NameNo.	CaEVNo.	ConnectDustVacuo	:=	61	;	//
NameNo.	CaEVNo.	LineSceneDustBlow	:=	62	;	//
NameNo.  CaEVNo.	LineSceneDustVacuo	:=	63	;	//
NameNo.	CaEVNo.	AreaArrayDustBlow	:=	64	;	//
NameNo.	CaEVNo.	MouldUpBlow	:=	65	;	//
NameNo.	CaEVNo.	MouldDownVacuo	:=	66	;	//
NameNo.	CaEVNo.	MouldDownAir	:=	67	;	//
NameNo.	CaEVNo.	NGPushInsideAir	:=	68	;	//
NameNo.	CaEVNo.	NGPushInsideVacuo	:=	69	;	//
NameNo.	CaEVNo.	BrushDustVacuo_U	:=	70	;	//
NameNo.	CaEVNo.	WindDustBlow_U	:=	71	;	//
NameNo.	CaEVNo.	WindDustVacuo_U	:=	72	;	//
NameNo.	CaEVNo.	BrushDustVacuo_D	:=	73	;	//
NameNo.	CaEVNo.	WindDustBlow_D	:=	74	;	//
NameNo.	CaEVNo.	WindDustVacuo_D	:=	75	;	//
NameNo.	CaEVNo.	RJ_Blow	:=	76	;	//
NameNo.	CaEVNo.	RJDustBlow	:=	77	;	//
						
	//////纠偏号//////					
NameNo.	AnRecNo.PoleWind:=1;(***极片放卷纠偏*)					
NameNo.	AnRecNo.PoleProcess:=2;(***极片行进纠偏*)					
						
NameNo.	CaRecNo.PoleWind:=3;(***极片放卷纠偏*)					
NameNo.	CaRecNo.PoleProcess:=4;(***极片行进纠偏*)					
						
	//////凸轮编号//////					
NameNo.	AnTableNo.	Cuter	:=	11	;(*裁切切刀凸轮编号*)	
NameNo.	AnTableNo.	CuterStop	:=	12	;(*裁切切刀停止凸轮编号*)	
NameNo.	AnTableNo.	Mould	:=13	;(*模具切刀凸轮编号*)		
NameNo.	AnTableNo.	MouldStop	:=14	;(*模具切刀停止凸轮编号*)		
NameNo.	AnTableNo.	Dirver	:=15	;(*主驱动凸轮编号*)		
NameNo.	AnTableNo.	VirBelt	:=	16	;(*虚拟皮带凸轮编号*)	
NameNo.	AnTableNo.	NgPush	:=	17	;(*NG踢料凸轮编号*)	
NameNo.	AnTableNo.	NgPushStop	:=	18	;(*NG踢料停止凸轮编号*)	
NameNo.	AnTableNo.	BufferLine	:=19	;(*极片缓存凸轮编号*)		
NameNo.	AnTableNo.	CCDPress	:=	20	;(*CCD压片凸轮编号*)	
NameNo.	AnTableNo.	BufferLine_1	:=	21	;(*极片缓存凸轮编号1*)	
NameNo.	AnTableNo.VirDirver	:=	22	;(*正极虚拟驱动凸轮编号1*)	
						
NameNo.	CaTableNo.	Cuter	:=	31	;(*裁切切刀凸轮编号*)	
NameNo.	CaTableNo.	CuterStop	:=	32	;(*裁切切刀停止凸轮编号*)	
NameNo.	CaTableNo.	Mould	:=	33	;(*模具切刀凸轮编号*)	
NameNo.	CaTableNo.	MouldStop	:=	34	;(*模具切刀停止凸轮编号*)	
NameNo.	CaTableNo.	Dirver	:=	35	;(*主驱动凸轮编号*)	
NameNo.	CaTableNo.	VirBelt	:=	36	;(*虚拟皮带凸轮编号*)	
NameNo.	CaTableNo.	NgPush	:=	37	;(*NG踢料凸轮编号*)	
NameNo.	CaTableNo.	NgPushStop	:=	38	;(*NG踢料停止凸轮编号*)	
NameNo.	CaTableNo.	BufferLine	:=	39	;(*极片缓存凸轮编号*)	
NameNo.	CaTableNo.	CCDPress	:=	40	;(*CCD压片凸轮编号*)	
NameNo.	CaTableNo.	BufferLine_1	:=	41	;(*极片缓存凸轮编号1*)					
NameNo.	CaTableNo.VirDirver	:=	42	;(*负极虚拟驱动凸轮编号1*)						
	//////皮带工位号//////					
NameNo.	AnBeltNo.	First	:=1	;	//	首片数据
NameNo.	AnBeltNo.	OverHang	:=2	;	//	尺寸检测工位
NameNo.	AnBeltNo.	NGBox1	:=4	;	//	踢废工位1（连续）
NameNo.	AnBeltNo.	NGBox2	:=6	;	//	踢废工位2（单片）
NameNo.	AnBeltNo.	BrushDustU	:=7	;	//	极片上表面毛刷除尘工位
NameNo.	AnBeltNo.	WindDustU	:=8	;	//	极片上表面风刀除尘工位
NameNo.	AnBeltNo.	BrushDustD	:=9	;	//	极片下表面毛刷除尘工位
NameNo.	AnBeltNo.	WindDustD	:=10	;	//	极片下表面风刀除尘工位(除尘倒装皮带末位)
NameNo.	AnBeltNo.	SubBelt1	:=14	;	//	分段皮带1取料工位
NameNo.	AnBeltNo.	SubBelt2	:=22	;	//	分段皮带2取料工位
NameNo.	AnBeltNo.	SubBelt3	:=30	;	//	分段皮带3取料工位
						
NameNo.	CaBeltNo.	First	:=1	;	//	首片
NameNo.	CaBeltNo.	OverHang	:=2	;	//	尺寸检测工位
NameNo.	CaBeltNo.	NGBox1	:=4	;	//	踢废工位1（连续）
NameNo.	CaBeltNo.	NGBox2	:=6	;	//	踢废工位2（单片）
NameNo.	CaBeltNo.	BrushDustU	:=7	;	//	极片上表面毛刷除尘工位
NameNo.	CaBeltNo.	WindDustU	:=8	;	//	极片上表面风刀除尘工位
NameNo.	CaBeltNo.	BrushDustD	:=9	;	//	极片下表面毛刷除尘工位
NameNo.	CaBeltNo.	WindDustD	:=10	;	//	极片下表面风刀除尘工位(除尘倒装皮带末位)
NameNo.	CaBeltNo.	SubBelt1	:=12	;	//	分段皮带1取料工位
NameNo.	CaBeltNo.	SubBelt2	:=20	;	//	分段皮带2取料工位
NameNo.	CaBeltNo.	SubBelt3	:=28	;	//	分段皮带3取料工位
						
	//////极耳工位号//////					
NameNo.	AnTabNo.MouldPhoto	:=1	;	//	倒角前拍照位置	
NameNo.	AnTabNo.CuterPhoto	:=6	;	//	裁切前拍照位置	
						
NameNo.	CaTabNo.MouldPhoto	:=1	;	//	倒角前拍照位置	
NameNo.	CaTabNo.CuterPhoto	:=6	;	//	裁切前拍照位置	
						
	//////极耳间距工位号//////					
NameNo.	AnIntervalNo.First	:=1	;	//	蓝胶位置	
NameNo.	AnIntervalNo.Mould	:=5	;	//	冲R角位置	
NameNo.	AnIntervalNo.Cuter	:=10	;	//	裁切位置	
						
NameNo.	CaIntervalNo.First	:=1	;	//	蓝胶位置	
NameNo.	CaIntervalNo.Mould	:=5	;	//	冲R角位置	
NameNo.	CaIntervalNo.Cuter	:=10	;	//	裁切位置	
						
	//////除尘电机号//////	
NameNo.	AnMotorNo.	DDR_Dust	:=	1	;	//主驱辊除尘				
NameNo.	AnMotorNo.	CuterBeltDust	:=	2	;	//裁切输送皮带除尘
NameNo.	AnMotorNo.	NGReverseBeltDust	:=	3	;	//踢废倒装皮带除尘
NameNo.	AnMotorNo.	DedustBeltDust	:=	4	;	//极片上表面除尘皮带除尘
NameNo.	AnMotorNo.	DedustReverseBeltDust	:=	5	;	//极片下表面除尘倒装皮带除尘
NameNo.	AnMotorNo.	PoleBrushDust_U	:=	6	;	//极片上表面毛刷除尘
NameNo.	AnMotorNo.	PoleBrushDust_D	:=	7	;	//极片下表面毛刷除尘
NameNo.	AnMotorNo.	FeduanbeltDust1	:= 15;//正极分段皮带1毛刷
NameNo.	AnMotorNo.	FeduanbeltDust2	:= 16;//正极分段皮带2毛刷
NameNo.	AnMotorNo.	FeduanbeltDust3	:= 17;//正极分段皮带3毛刷

NameNo.	CaMotorNo.	DDR_Dust	:=	8	;	//主驱辊除尘							
NameNo.	CaMotorNo.	CuterBeltDust	:=	9	;	//裁切输送皮带除尘
NameNo.	CaMotorNo.	NGReverseBeltDust	:=	10	;	//踢废倒装皮带除尘
NameNo.	CaMotorNo.	DedustBeltDust	:=	11	;	//极片上表面除尘皮带除尘
NameNo.	CaMotorNo.	DedustReverseBeltDust	:=	12	;	//极片下表面除尘倒装皮带除尘
NameNo.	CaMotorNo.	PoleBrushDust_U	:=	13	;	//极片上表面毛刷除尘
NameNo.	CaMotorNo.	PoleBrushDust_D	:=	14	;	//极片下表面毛刷除尘
NameNo.	CaMotorNo.	FeduanbeltDust1	:=	18	;	//负极分段皮带1毛刷
NameNo.	CaMotorNo.	FeduanbeltDust2	:=	19	;	//负极分段皮带2毛刷
NameNo.	CaMotorNo.	FeduanbeltDust3	:=	20	;	//负极分段皮带3毛刷

IF ProductPar.parPublic.fMainPos <>250 THEN
	ProductPar.parPublic.fMainPos:=250;
END_IF
IF ProductPar.AnPar.fPoleWidth=0 THEN
	ProductPar.AnPar.fPoleWidth:=186;
END_IF
IF ProductPar.CaPar.fPoleWidth=0 THEN
	ProductPar.CaPar.fPoleWidth:=188;
END_IF
IF ProductPar.AnPar.Machine.fMQDriverDiameter=0 THEN
	ProductPar.AnPar.Machine.fMQDriverDiameter:=71.62;
END_IF
IF ProductPar.CaPar.Machine.fMQDriverDiameter=0 THEN
	ProductPar.CaPar.Machine.fMQDriverDiameter:=71.62;
END_IF
IF ProductPar.AnPar.iMainVel=0 THEN
	ProductPar.AnPar.iMainVel:=10;
END_IF
IF ProductPar.CaPar.iMainVel=0 THEN
	ProductPar.CaPar.iMainVel:=10;
END_IF


(***DDR位置上电清零***)
arrAxisCtrl[NameNo.AnAxisNo.DriverDDR].Cmd.fSetPos:=360;
arrAxisCtrl[NameNo.AnAxisNo.DriverDDR].Cmd.bSetPos:=TRUE;

arrAxisCtrl[NameNo.CaAxisNo.DriverDDR].Cmd.fSetPos:=360;
arrAxisCtrl[NameNo.CaAxisNo.DriverDDR].Cmd.bSetPos:=TRUE;

IF arrAxisCtrl[NameNo.AnAxisNo.DriverDDR].Cmd.fSetPos>=0 AND arrAxisCtrl[NameNo.CaAxisNo.DriverDDR].Cmd.fSetPos>=0 THEN
	arrAxisCtrl[NameNo.AnAxisNo.DriverDDR].Cmd.bSetPos:=FALSE;
	arrAxisCtrl[NameNo.CaAxisNo.DriverDDR].Cmd.bSetPos:=FALSE;
	iPowerSetp:=666;
	PowerOnDone:=TRUE;
END_IF
//////////////////////////////////////////////////////////////

END_CASE
 
bytePower.0;
bytePower.1;
bytePower.2;
bytePower.3;
bytePower.4;
bytePower.5;
bytePower.6;
bytePower.7;
END_ACTION

ACTION TwinCAT_Nt:
//fPlcCycleTime_ms:=UDINT_TO_LREAL(_TaskInfo[0].CycleTime)/10000;

(***********************  保存掉电保持数据   **************************************)
tCycleTimer(IN:=NOT tCycleTimer.Q , PT:=T#356S , Q=>bWrite , ET=> );
rt[1](CLK:=tCycleTimer.ET>=T#1M , Q=>bWrite );
FB_WritePersistentData1(
	NETID:='' ,
	PORT:=851 ,
	START:=bWrite OR  stHmiSysCmd.bSaveData  ,//OR    _TaskInfo[1].FirstCycle 
	TMOUT:=t#500ms ,
	MODE:=SPDM_2PASS ,
	BUSY=>BUSY ,
	ERR=> ERR,
	ERRID=>ERRID );
ft[1](CLK:=BUSY , Q=> );
IF ft[1].Q THEN
	bDataValid:=TRUE;
END_IF	
	
	
	
(********************** 获取系统时间   ***************************************)
NT_GetTime1(
	NETID:='' ,
	START:=Pulse._1s.RT ,
	TMOUT:= ,
	BUSY=> ,
	ERR=> ,
	ERRID=> ,
	TIMESTR=>stTime );

	strTime:=CONCAT(CONCAT(CONCAT(CONCAT(CONCAT(CONCAT(CONCAT(CONCAT( CONCAT(CONCAT( WORD_TO_STRING(stTime.wYear),'-'), WORD_TO_STRING(stTime.wMonth)),'-'),WORD_TO_STRING(stTime.wDay)),
             '-'),WORD_TO_STRING(stTime.wHour)),'-'),WORD_TO_STRING(stTime.wMinute)),'-'),WORD_TO_STRING(stTime.wSecond));
	

	PLC_wYear:=stTime.wYear;//PLC时间年
	PLC_wMonth:=stTime.wMonth;//PLC时间月
	PLC_wDay:=stTime.wDay;//PLC时间日
	PLC_wHour:=stTime.wHour;//PLC时间时
	PLC_wMinute:=stTime.wMinute;//PLC时间分
	PLC_wSecond:=stTime.wSecond;//PLC时间秒	
	PLC_wMilliseconds:=stTime.wMilliseconds;//PLC时间秒	
		 

(********************************** Systemfunctions **********************************************************)
	SysInfo(
		Reset				:= ,
		TimeStampTrig		:= Pulse._100ms.RT,
		//RunTimeNo			=> ,
		//ProjectName			=> ,
		//NumberOfTasks		=> ,
		//OnlineChangeCount	=> ,
		RetainVarErr		=> ,
		PersistenVarErr		=> ,
		TimeStampDT			=> ,
		TimeStamp			=> ,
		TimeStr				=> ,
		DateStr				=> ,
		TimeStamp2			=> ,
		TimeStruct			=> ,
		MonthDays			=> ,
		LeapYear			=> ,
		WeekOfYear			=> ,
		timezoneId			=>);

	TaskInfo(
		index				=> ,
		active				=> ,
		taskName			=> ,
		firstCycle			=> ,
		cycleTimeExceeded	=> ,
		cycleTime			=> ,
		lastExecTime		=> ,
		priority			=> ,
		cycleCount			=> );

	Pulse(
		BlinkSlow			=> ,
		Blink				=> ,
		BlinkFast			=> );	
		
	(*系统重启，CE远程桌面，系统时间，定时保存掉电数据，等系统常规动作*)
(**********************  通讯心跳信号   ***************************************)
TonHeartBeat(IN:=NOT TonHeartBeat.Q , PT:=tHeartBeatTime , Q=> , ET=> );
IF TonHeartBeat.Q THEN
	bHeartBeat:=NOT bHeartBeat;
END_IF

tNtDelayReset(IN:=stHmiSysCmd.bRebootPc OR bReboot , PT:=T#1S , Q=> , ET=> );
NT_Reboot1(
	NETID:='' ,
	DELAY:= ,
	START:=tNtDelayReset.Q  ,
	TMOUT:=DEFAULT_ADS_TIMEOUT ,
	BUSY=> ,
	ERR=> ,
	ERRID=> );

tNtDelayShutdown(IN:=stHmiSysCmd.bShutDownPc OR bShutDown , PT:=T#1S , Q=> , ET=> );	(*触摸屏上已经做了延时*)
NT_Shutdown1(
	NETID:= ,
	DELAY:= ,
	START:=tNtDelayShutdown.Q,
	TMOUT:=DEFAULT_ADS_TIMEOUT ,
	BUSY=> ,
	ERR=> ,
	ERRID=> );
END_ACTION

ACTION XML:

IF NOT  bReadDataFirstCyle THEN //testii:=testii+1;
	//fbDataXML.bRead:=NOT bDataValid;
	bReadDataFirstCyle:=TRUE;
END_IF


IF fbDataXML.bReadParDone AND bReadDataFirstCyle   AND   NOT bReadDataCyle2      THEN
	PoleData:= ProductPar.PoleData;
	YL_GVL2:=ProductPar.YL_GVL2;
	iTargetTorque:=ProductPar.iTargetTorque;
	bReadDataCyle2:=TRUE;
END_IF
	 


rt[2](CLK:=tCycleTimer.ET>=T#2M , Q=> );
rtSaveData(CLK:=stHmiSysCmd.bSaveData , Q=> );
IF  rtSaveData.Q THEN
	bSaveTest:=TRUE;
END_IF


IF  rt[2].Q  OR bSaveTest THEN
	ProductPar.PoleData:=PoleData  ;
	ProductPar.YL_GVL2 :=YL_GVL2  ;
	ProductPar.iTargetTorque:=iTargetTorque   ;	 
	bSaveTest:=FALSE;
	fbDataXML.bSave:=TRUE;
	testii2:=testii2+1;
END_IF

rt[4](CLK:=stHmiSysCmd.bReadData (*AND  stSysState.iMode=3*), Q=> );
rt[5](CLK:=PowerOnDone , Q=> );
tRead(IN:=PowerOnDone, PT:=T#3S , Q=> , ET=> );
IF   tRead.Q AND NOT fbDataXML.bReadParDone THEN
	  breadALM:=TRUE;//上电后模切参数读取失败，请手动点读取参数
END_IF

IF  stSysState.bReset THEN
	 breadALM:=FALSE;
END_IF
fbDataXML(bSave:=fbDataXML.bSave AND NOT breadALM, bRead:=fbDataXML.bRead OR rt[4].Q OR rt[5].Q, bSaveParDone=> , bReadParDone=> );

fbDataXML.bReadParDone;
fbDataXML.bSaveParDone;

(*
//fbPulseCtrl[7](PT_OFF:=T#30M, PT_ON:=T#30M, );
//fbPulseCtrl[7].Q;
//fbPulseCtrl[7].RT;


tCycleTimer(IN:=NOT tCycleTimer.Q , PT:=T#311S , Q=>bSave , ET=> );
rt10(clk:=bSave);
IF NOT  bReadDataFirstCyle THEN //testii:=testii+1;
	 	 fbDataXML.bRead:=TRUE;
	     testii:=testii+1;
	    bReadDataFirstCyle:=TRUE;
		
END_IF


IF fbDataXML.bReadParDone AND bReadDataFirstCyle   AND   NOT bReadDataCyle2      THEN
     aAnDay_date:=ProductPar.aAnDay_date;
     aCaDay_date:=ProductPar.aCaDay_date;
     cCn_An:=ProductPar.cCn_An;
     cCn_Ca:=ProductPar.cCn_Ca;
	 PoleData:= ProductPar.PoleData;
	 
     YL_GVL2:=ProductPar.YL_GVL2;
	 
     HMI_AnTodayNGClass_AM:=ProductPar.HMI_AnTodayNGClass_AM;
     HMI_AnTodayNGClass_PM:=ProductPar.HMI_AnTodayNGClass_PM;
     HMI_AnTodayNG_AM:=ProductPar.HMI_AnTodayNG_AM;
     HMI_AnTodayNG_PM:=ProductPar.HMI_AnTodayNG_PM;
     HMI_CaTodayNGClass_AM:=ProductPar.HMI_CaTodayNGClass_AM;
     HMI_CaTodayNGClass_PM:=ProductPar.HMI_CaTodayNGClass_PM;
     HMI_CaTodayNG_AM:=ProductPar.HMI_CaTodayNG_AM;
     HMI_CaTodayNG_PM:=ProductPar.HMI_CaTodayNG_PM;
	  iTargetTorque:=ProductPar.iTargetTorque;
	 

	 bReadDataCyle2:=TRUE;
  END_IF
	 



rtSaveData(CLK:=stHmiSysCmd.bSaveData , Q=> );
IF  rtSaveData.Q THEN
	bSaveTest:=TRUE;
END_IF


IF  rt10.Q  OR bSaveTest    THEN
     ProductPar.aAnDay_date:=aAnDay_date   ;
     ProductPar.aCaDay_date:=aCaDay_date ;
     ProductPar.cCn_An:=cCn_An   ;
     ProductPar.cCn_Ca:=cCn_Ca  ;
	 ProductPar.PoleData:=PoleData  ;
	 
     ProductPar.YL_GVL2 :=YL_GVL2  ;
	 
     HMI_AnTodayNGClass_AM := ProductPar.HMI_AnTodayNGClass_AM   ;
     HMI_AnTodayNGClass_PM:=ProductPar.HMI_AnTodayNGClass_PM  ;                      ;
     ProductPar.HMI_AnTodayNG_AM :=HMI_AnTodayNG_AM  ;
     ProductPar.HMI_AnTodayNG_PM:=HMI_AnTodayNG_PM   ;
     ProductPar.HMI_CaTodayNGClass_AM:=HMI_CaTodayNGClass_AM   ;
     ProductPar.HMI_CaTodayNGClass_PM:=HMI_CaTodayNGClass_PM ;
     ProductPar.HMI_CaTodayNG_AM:=HMI_CaTodayNG_AM   ;
     ProductPar.HMI_CaTodayNG_PM:=HMI_CaTodayNG_PM   ;	 
     ProductPar.iTargetTorque:=iTargetTorque   ;	 

     bSaveTest:=FALSE;
	fbDataXML.bSave:=TRUE;
	testii2:=testii2+1;
END_IF

fbDataXML(bSave:=fbDataXML.bSave AND D_Sys.P3ReadParDone, 
                     bRead:=fbDataXML.bRead , 
                     bSaveParDone=> ,
                     bReadParDone=> );
					 

M_Sys.P1ReadParDone:=fbDataXML.bReadParDone;
M_Sys.P1SaveParDone:=fbDataXML.bSaveParDone;
*)
END_ACTION

END_PROGRAM

// ---- POUs/BasicFunction/Data/CS_Data.TcPOU
FUNCTION_BLOCK CS_Data
VAR_INPUT
END_VAR
VAR_OUTPUT
END_VAR
VAR
	//tDataSave:TON;
	//fbSaveData:FB_WritePersistentData;
	//fbXMLWrite:FB_XMLSrvWrite;
	//bWriteXml: BOOL;
	
	fbFileOpen_w:fb_fileopen;
	//fbFileOpen_r:fb_fileopen;
	fbFileWrite:fb_filewrite;
	fbFileRead:FB_FileRead;
	fbFileClose_w:fb_FileClose;
	//fbFileClose_r:fb_FileClose;
	HFILE:UINT;
	//HFILE_R:UINT;
	//bFileOpen_w:BOOL;
	//bFileOpen_r:BOOL;
	//bFileWrite:BOOL;
	//bFileClose_w:BOOL;
	//bFileClose_r:BOOL;
	//bFileRead:BOOL;
	bSave:BOOL;
	bRead:BOOL;
//	tFileOper_Save:TON;
	//tFileOper_Read:TON;
	iDataSetp: INT;
	TON10:Tc2_Standard.TON;
	bExecute: BOOL;
	I1: INT;
	rt100:Tc2_Standard.R_TRIG;
	rt101:Tc2_Standard.R_TRIG;
	bExecute1: BOOL;
	bExecute2: BOOL;
	bExecute3: BOOL;	

	bSaveTemp: BOOL;
	bReadTemp: BOOL;
	bReadDataOk: BOOL;
END_VAR


M_WriteOrRead();

ACTION M_WriteOrRead:


(*
rt100(CLK:=bSave , Q=> );//保存参数
rt101(CLK:=bRead , Q=> );//读取参数

IF rt100.Q THEN
	iDataSetp:=100;
	TON10.IN:=FALSE;
	I1:=1;
	bExecute1:=FALSE;
	bExecute2:=FALSE;	
	bExecute3:=FALSE;	
	bSave:=FALSE;
	bRead:=FALSE;
    bSaveTemp:=TRUE;
	bReadTemp:=FALSE;
END_IF

IF rt101.Q THEN
	iDataSetp:=100;
	TON10.IN:=FALSE;
	I1:=1;
	bExecute1:=FALSE;
	bExecute2:=FALSE;	
	bExecute3:=FALSE;	
	bSave:=FALSE;
	bRead:=FALSE;
    bReadTemp:=TRUE;
    bSaveTemp:=FALSE;
END_IF

TON10(IN:= , PT:=T#200MS , Q=> , ET=> );
//保存配方	
CASE  iDataSetp OF 
	
	100:	//参数给定
	   
	   IF bSaveTemp THEN
	     fbFileOpen_w.nMode:=FOPEN_MODEWRITE OR FOPEN_MODEBINARY;
	   END_IF
	   IF bReadTemp THEN
	     fbFileOpen_w.nMode:=FOPEN_MODEREAD OR  FOPEN_MODEBINARY;
	   END_IF
	  iDataSetp:=101;
	101:

	  CASE I1 OF 
		1:
		 fbFileWrite.pWriteBuff:=ADR(gstM1Par);
		 fbFileWrite.cbWriteLen:=SIZEOF(gstM1Par);
		 fbFileRead.pReadBuff:=ADR(gstM1Par1);
		 fbFileRead.cbReadLen:=SIZEOF(gstM1Par1);
		 fbFileOpen_w.sPathName:='C:\P2Data\M1.bin';
		2:
		 fbFileWrite.pWriteBuff:=ADR(gstM2Par);
		 fbFileWrite.cbWriteLen:=SIZEOF(gstM2Par);
		 fbFileRead.pReadBuff:=ADR(gstM2Par1);
		 fbFileRead.cbReadLen:=SIZEOF(gstM2Par1);
		 fbFileOpen_w.sPathName:='C:\P2Data\M2.bin';
		3:
		 fbFileWrite.pWriteBuff:=ADR(gstM3Par);
		 fbFileWrite.cbWriteLen:=SIZEOF(gstM3Par);
		 fbFileRead.pReadBuff:=ADR(gstM3Par1);
		 fbFileRead.cbReadLen:=SIZEOF(gstM3Par1);
		 fbFileOpen_w.sPathName:='C:\P2Data\M3.bin';
		4:
		 fbFileWrite.pWriteBuff:=ADR(gstM4Par);
		 fbFileWrite.cbWriteLen:=SIZEOF(gstM4Par);
		 fbFileRead.pReadBuff:=ADR(gstM4Par1);
		 fbFileRead.cbReadLen:=SIZEOF(gstM4Par1);
		 fbFileOpen_w.sPathName:='C:\P2Data\M4.bin';
		5:  
		 fbFileWrite.pWriteBuff:=ADR(gstM5Par);
		 fbFileWrite.cbWriteLen:=SIZEOF(gstM5Par); 
		 fbFileRead.pReadBuff:=ADR(gstM5Par1);
		 fbFileRead.cbReadLen:=SIZEOF(gstM5Par1);
		 fbFileOpen_w.sPathName:='C:\P2Data\M5.bin';
	  END_CASE
	  iDataSetp:=200;
	
	200:	//打开文件
		bExecute1:=TRUE;
		TON10.IN:=TRUE;
	  IF TON10.Q THEN
		 bExecute1:=FALSE; 
		 TON10.IN:=FALSE;
		 iDataSetp:=300; 
	  END_IF
	
	300:	//读写文件
		bExecute2:=TRUE;
		TON10.IN:=TRUE;
	  IF TON10.Q THEN
		  bExecute2:=FALSE; 
		  TON10.IN:=FALSE;
		 iDataSetp:=400; 
	  END_IF
	
	400:	//关闭文件
		bExecute3:=TRUE;
		TON10.IN:=TRUE;
	  IF TON10.Q THEN
		  bExecute3:=FALSE; 
		  TON10.IN:=FALSE;
		  iDataSetp:=500; 
	  END_IF
	
	500://继续写下个文件
	  IF I1>=1 AND I1<5 THEN
		 I1:=I1+1; 
		 TON10.IN:=FALSE;
		 iDataSetp:=100; 
		 bExecute1:=FALSE; 
		 bExecute2:=FALSE; 
		 bExecute3:=FALSE; 
	  ELSIF I1>=5 THEN
		  bReadTemp:=FALSE;
          bSaveTemp:=FALSE;
		 iDataSetp:=666;   
	  END_IF
END_CASE


IF bReadDataOk THEN
   gstM1Par:=gstM1Par1;
   gstM2Par:=gstM2Par1;
   gstM3Par:=gstM3Par1;
   gstM4Par:=gstM4Par1;	
   gstM5Par:=gstM5Par1;
   bReadDataOk:=FALSE;
END_IF










   	fbFileOpen_w(
	sNetId:= , 
	sPathName:= , //C:\P2Data
	nMode:=   , 
	ePath:=PATH_GENERIC , 
	bExecute:=bExecute1 , 
	tTimeout:=T#3S , 
	bBusy=> , 
	bError=> , 
	nErrId=> , 
	hFile=>hfile );


	fbFileWrite(
	sNetId:= , 
	hFile:= hFile, 
	pWriteBuff:= , 
	cbWriteLen:= , 
	bExecute:=bExecute2 AND bSaveTemp, 
	tTimeout:=T#3S , 
	bBusy=> , 
	bError=> , 
	nErrId=> , 
	cbWrite=> );



	fbFileRead(
	sNetId:= , 
	hFile:=hFile , 
	pReadBuff:= , 
	cbReadLen:= , 
	bExecute:= bExecute2 AND bReadTemp, 
	tTimeout:= T#3S, 
	bBusy=> , 
	bError=> , 
	nErrId=> , 
	cbRead=> , 
	bEOF=> );


	fbFileClose_w(
	sNetId:= , 
	hFile:= hFile, 
	bExecute:= bExecute3, 
	tTimeout:=T#3S , 
	bBusy=> , 
	bError=> , 
	nErrId=> );
	
	
	
*)
END_ACTION

END_FUNCTION_BLOCK

// ---- POUs/BasicFunction/SystemInfo/TaskInfoCtrl.TcPOU
FUNCTION_BLOCK TaskInfoCtrl
VAR_INPUT
END_VAR
VAR_OUTPUT
	index						:	INT;
	active					:	BOOL; 		(* Diese Variable zeigt an, ob die Task aktiv ist.*)
	taskName					:	STRING(16);	(* Der Taskname.*)
	firstCycle				:	BOOL;			(* Diese Variable hat im ersten Zyklus der SPS-Task den Wert: TRUE.*)
	cycleTimeExceeded		:	BOOL;			(* In dieser Variablen wird ein 躡erschreiten der eingestellten Taskzykluszeit gemeldet*)
	cycleTime				:	UDINT;		(* Eingestellte Taskzykluszeit in Vielfachen von 100ns*)
	lastExecTime			:	UDINT;		(* Ben鰐igte Zykluszeit f黵 den letzten Zyklus in Vielfachen von 100 ns*)
	MaxExecTime				:	UDINT;		(* Maximale Zykluszeit *)
	priority					:	BYTE;			(* Eingestellte Prioritaet der Task*)
	cycleCount				: 	UDINT;		(* Zykluszaehler*)
END_VAR

VAR
	GETCURTASKINDEX		: GETCURTASKINDEX;
END_VAR

	(*********************************************************************************)
	(*	(c) by Beckhoff Automation																		*)
	(*																											*)
	(*		B E C K H O F F   N E W   A U T O M A T I O N   T E C H N O L O G Y        *)
	(*																											*)
	(*		Eiserstr.5	D-33415 Verl	Germany	phone:	+49-5246-0	www.Beckhoff.com	*)
   (*																											*)
   (*		Bausteinbeschreibung	: Auswerten des SystemInfoTaskArrays 						*)
	(*																											*)
	(*		Version				:	V1.0																	*)
	(*		Stand					:	04.2009																*)
 	(*		Autor					:	Daniel Schlingmann												*)
	(*																											*)
	(*********************************************************************************)

(* Get Current Task Index ************************************************************************)
	GETCURTASKINDEX(index => index);

	(* Retein/Persisten Data Err *)
	//active :=  _TaskInfo[index].active;
	taskName :=  _TaskInfo[index].TaskName;
	firstCycle :=  _TaskInfo[index].FirstCycle;
	cycleTimeExceeded :=  _TaskInfo[index].CycleTimeExceeded;
	cycleTime :=  _TaskInfo[index].CycleTime;
	lastExecTime :=  _TaskInfo[index].LastExecTime;
	MaxExecTime	:= MAX(lastExecTime,MaxExecTime);
//	priority :=  _TaskInfo[index].Priority;
	firstCycle :=  _TaskInfo[index].FirstCycle;
	cycleCount :=  _TaskInfo[index].CycleCount;

(**************************************************************************************************)

END_FUNCTION_BLOCK

// ---- POUs/BasicFunction/User1/FB_DataXML.TcPOU
FUNCTION_BLOCK FB_DataXML
VAR_INPUT
    	bSave:BOOL;
	    bRead:BOOL;
		bReadSel:BOOL;//参数读取选择，TRUE=选择恢复上电备份的参数
END_VAR
VAR_OUTPUT
    	bSaveParDone      :BOOL;
	    bReadParDone     :BOOL;
END_VAR

VAR
	iDataSetp: INT;
	i1: INT;
	i2:BYTE;
	rt100:Tc2_Standard.R_TRIG;
	rt101:Tc2_Standard.R_TRIG;
	rt102:Tc2_Standard.R_TRIG;
	rt103:Tc2_Standard.R_TRIG;
	bSaveTemp: BOOL;
	bReadTemp: BOOL;
	sFilePath:STRING;//文件路径
	sNewFilePath:STRING;//新文件路径
	sOldFilePath:STRING;//旧文件路径
	sFileName:STRING;//文件名称
	sVarName:STRING;//变量名称
	fbXmlSrvRead				: FB_XmlSrvReadByName;//读取XML文件	
	fbXmlSrvWrite				: FB_XmlSrvWriteByName;//写入XML文件
	bFirstCycleFlg:BOOL;//首次执行标志位
	fbGetFileList: FB_GetFileList;//获取文件列表功能块
	stFindFileEntry:ARRAY[1..50] OF ST_FindFileEntry;//文件列表存放结构体	
	nFileBakStep:UINT;//文件备份步序
	fbFileDelete	: FB_FileDelete;//删除文件
	fbFileRename	: FB_FileRename;//文件重命名
	fbCreateDirectory:FB_CreateDirectory;//文件夹创建
END_VAR

M_WriteOrRead();
A_FileBak();

ACTION A_FileBak:
CASE nFileBakStep OF
	200:
		fbGetFileList(bExecute:=FALSE);
		fbFileDelete(bExecute:=FALSE);
		fbFileRename(bExecute:=FALSE);
		fbCreateDirectory(bExecute:=FALSE);
		nFileBakStep:=300;
	300:(*获取文件列表*)
		fbGetFileList.pFindFileListADR:=ADR(stFindFileEntry);
		fbGetFileList.u32FindFileListSizeOf:=SIZEOF(stFindFileEntry);
		fbGetFileList(bExecute:=TRUE,sgPathName:=sOldFilePath,sgFileType:='xml');	
		IF fbGetFileList.bDone THEN
			fbGetFileList(bExecute:=FALSE);
			nFileBakStep:=310;
		ELSIF fbGetFileList.bError THEN
			fbGetFileList(bExecute:=FALSE);
			nFileBakStep:=997;
		END_IF
	310:(*判断文件是否存在，文件存在则备份一次，文件不存在直接给完成信号*)
		FOR i2:=1 TO 50 DO
			IF stFindFileEntry[i2].sFileName=sFileName THEN//
				EXIT;
			END_IF
		END_FOR
		IF i2>50 THEN
			nFileBakStep:=666;
		ELSE
			nFileBakStep:=320;
		END_IF
	320:(*文件夹创建*)
	fbCreateDirectory(bExecute:=TRUE , sgPathName:=sNewFilePath, tTimeout:=T#1S );
	IF fbCreateDirectory.bDone THEN
		fbCreateDirectory(bExecute:=FALSE);
		nFileBakStep:=350;
	ELSIF fbCreateDirectory.bError THEN
		fbCreateDirectory(bExecute:=FALSE);
		nFileBakStep:=998;
	END_IF
	350:(*删除旧文件*)
		fbFileDelete.sPathName:= CONCAT(sNewFilePath,sFileName);
		fbFileDelete(bExecute:=TRUE,ePath:= PATH_GENERIC,tTimeout:=T#5S);
		IF NOT fbFileDelete.bBusy THEN
			fbFileDelete(bExecute:=FALSE);
			nFileBakStep:=360;
		END_IF
	360:(*重命名文件*)
		fbFileRename.sOldName:= CONCAT(sOldFilePath,sFileName);
		fbFileRename.sNewName:= CONCAT(sNewFilePath,sFileName);
		fbFileRename(bExecute:=TRUE,ePath:= PATH_GENERIC,tTimeout:=T#5S);
		IF NOT fbFileRename.bBusy THEN
			fbFileRename(bExecute:=FALSE);
			IF NOT fbFileRename.bError THEN
				nFileBakStep:=666;
			ELSE
				nFileBakStep:=999;
			END_IF			
		END_IF
END_CASE
END_ACTION

ACTION M_WriteOrRead:
rt100(CLK:=bSave , Q=> );//保存参数
rt101(CLK:=bRead , Q=> );//读取参数
IF rt100.Q THEN  //保存参数
    bSaveTemp:=TRUE;
	bReadTemp:=FALSE;
	bSaveParDone:=FALSE;
	iDataSetp:=50;
END_IF
IF rt101.Q THEN  //读取参数
    bReadTemp:=TRUE;
    bSaveTemp:=FALSE;
	bReadParDone:=FALSE;
	iDataSetp:=50;
END_IF

//rt102(CLK:=NOT bFirstCycleFlg AND NOT bReadTemp, Q=> );//首次上电自动备份参数
IF rt102.Q THEN  //首次上电自动备份参数
	iDataSetp:=50;
END_IF

CASE  iDataSetp OF 
	50:
		I1:=1;
		fbXmlSrvRead(bExecute:=FALSE);
		fbXmlSrvWrite(bExecute:=FALSE);
		bSave:=FALSE;
		bRead:=FALSE;
		iDataSetp:=100;
	 100:
	 	sFilePath:='C:\P1XML\';//保存文件路径
		CASE i1 OF 
			 1://轴参数
				sFileName:= 'P1arrAxisPar.xml';
				sVarName:='GMotion.arrAxisPar';
			 2://ProductPar
				sFileName:='P1ProductPar.xml';
				sVarName:='GVL_Par.ProductPar';
			3://AnStats
				sFileName:='An_Production.xml';
				sVarName:='User01.An_Production';
			4://CaStats
				sFileName:= 'Ca_Production.xml';
				sVarName:='User01.Ca_Production';
		END_CASE		
		
		IF  bSaveTemp THEN
			iDataSetp:=200;
		ELSIF  bReadTemp THEN
			iDataSetp:=300;
		//ELSIF NOT bFirstCycleFlg THEN
		//	iDataSetp:=400;
		END_IF
		
	(********************保存数据流程：先备份原来参数再保存新参数，如果保存失败恢复至备份参数********************)
	200:(*开始备份*)
		sNewFilePath:=CONCAT(sFilePath,'Tmp\');
		sOldFilePath:=sFilePath;
		nFileBakStep:=200;//调用A_FileBak()进行文件备份
		iDataSetp:=210;
	210:(*文件备份状态判断*)
		IF nFileBakStep=666 THEN//文件备份成功，保存新参数
			iDataSetp:=230;
		ELSIF nFileBakStep>990 THEN//文件备份失败
			iDataSetp:=997;			
		END_IF
	230:(*保存新参数*)	
		fbXmlSrvWrite(
			bExecute:= TRUE, 
			ePath:=PATH_GENERIC , 
			nMode:=XMLSRV_ADDMISSING , 
			sSymName:=sVarName , 
			sFilePath:= CONCAT(sFilePath,sFileName), 
			sXPath:= '/DataEntry/Value', 
			tTimeout:= T#2S);
		IF NOT fbXmlSrvWrite.bBusy THEN
			fbXmlSrvWrite(bExecute:=FALSE);
			IF NOT fbXmlSrvWrite.bError THEN(*保存新参数成功*)
				iDataSetp:=500;
			ELSE(*保存新参数失败，恢复未写入新参数前的备份*)
				iDataSetp:=250;
			END_IF	
		END_IF
	250:(*保存新参数失败，恢复未写入新参数前的备份*)
		sOldFilePath:=CONCAT('Tmp\' ,sFileName);
		sNewFilePath:=sFilePath;
		nFileBakStep:=200;//调用A_FileBak()进行文件备份
		iDataSetp:=260;
	260:(*恢复文件状态判断*)
		IF nFileBakStep=666 THEN//文件恢复成功
			iDataSetp:=500;
		ELSIF nFileBakStep>990 THEN//文件恢复失败
			iDataSetp:=998;			
		END_IF		

	(********************参数读取流程********************)	
	300:(*参数读取选择，TRUE=选择恢复上电备份的参数*)
		IF bReadSel THEN
			sFilePath:=CONCAT(sFilePath,'Bak\');
		END_IF
		iDataSetp:=310;
	310:(*读取参数*)
		fbXmlSrvRead(
			bExecute:= TRUE, 
			ePath:=PATH_GENERIC , 
			nMode:=XMLSRV_ADDMISSING , 
			sSymName:= sVarName, 
			sFilePath:=CONCAT(sFilePath,sFileName) , 
			sXPath:='/DataEntry/Value' , 
			tTimeout:=T#2S);
		IF NOT fbXmlSrvRead.bBusy THEN
			fbXmlSrvRead(bExecute:=FALSE);
			IF NOT fbXmlSrvRead.bError THEN
				iDataSetp:=500;//读取成功
			ELSE
				iDataSetp:=999;//读取失败
			END_IF
		END_IF
		
	(********************上电自动备份流程，防止被覆盖********************)	
	400:
		sOldFilePath:=sFilePath;
		sNewFilePath:=CONCAT(sFilePath,'Bak\' );
		nFileBakStep:=200;//调用A_FileBak()进行文件备份
		iDataSetp:=410;
	410:
		IF nFileBakStep=666 THEN
				iDataSetp:=500;
		ELSIF nFileBakStep>990 THEN
				iDataSetp:=999;			
		END_IF
	500:(*继续写下个文件*)
		IF i1>=1 AND i1<4 THEN
			i1:=i1+1; 
			iDataSetp:=100; 
		ELSIF i1>=4 THEN
			IF  bSaveTemp THEN		
				bSaveParDone:=TRUE;
			ELSIF  bReadTemp THEN
				bReadParDone:=TRUE;
			ELSIF NOT bFirstCycleFlg THEN
				bFirstCycleFlg:=TRUE;
			END_IF
			bReadSel:=FALSE;
			bReadTemp:=FALSE;
			bSaveTemp:=FALSE;
			iDataSetp:=666;   
		END_IF
END_CASE
END_ACTION

END_FUNCTION_BLOCK

// ---- POUs/POUs/IOLink.TcPOU
PROGRAM IOLink
VAR
//	tFlash: TON;
//	bFlash:BOOL;
//	bIOinit: BOOL;
	XXX: INT;
	Q20815: BOOL;
	AA: INT;

     arrFilter_AD               : ARRAY[1..MaxAINo]  OF  FB_Filter_AD ;

      arrFilter_ADV2               : ARRAY[1..2]  OF  FB_Filter_ADV2 ;

	I1: INT;

    rt01   :Tc2_Standard.R_TRIG;
    rt02   :Tc2_Standard.R_TRIG;

     parDAOld                   :ARRAY[1..8] OF INT;   
	test1: BOOL;
END_VAR



InPut();

OutPut();

AI();

LimitSwitch();

IF fbPulseCtrl[4].RT THEN
      AO();
END_IF
(*
rt01(CLK:=arrCyCtrl[P3CYNo.RollPress].Cmd.bON , Q=> );
rt02(CLK:=arrCyCtrl[P3CYNo.RollPress].Cmd.bOFF , Q=> );
IF rt01.Q THEN
    P3EL4004S[3,1]:=parDA[33]	 ;//重力补偿
  //  P3EL4004S[3,2]:=parDA[34]	 ;
END_IF
IF rt02.Q THEN
    P3EL4004S[3,1]:=22000;//重力补偿
 //   P3EL4004S[3,2]:=20000;
END_IF
*)
//正极数据IOLink
ProductPar.AnPar.fSpeed:=GVL_Par.ProductPar.AnPar.iMainVel;
ProductPar.AnPar.fTension:=ProductPar.parFilterAD[3].Out_Value;

//负极数据IOLink
ProductPar.CaPar.fSpeed:=GVL_Par.ProductPar.CaPar.iMainVel;
ProductPar.CaPar.fTension:=ProductPar.parFilterAD[15].Out_Value;

ACTION AI:

//正极
arrFilter_AD[1].AD	:=	AI101[0];//	正极左放卷卷径超声波检测
arrFilter_AD[2].AD	:=	AI101[1];//	正极右放卷卷径超声波检测
//arrFilter_AD[3].AD	:=	AI101[2];//	正极辅驱前料带张力检测
arrFilter_ADV2[1].AD	:=	AI101[2];//	正极辅驱前料带张力检测
arrFilter_AD[4].AD	:=	AI101[3];//	备用
			
arrFilter_AD[5].AD	:=	AI102[0];//	正极后摆杆电位计检测
arrFilter_AD[6].AD	:=	AI102[1];//	正极倒角深度前纠偏检测
arrFilter_AD[7].AD	:=	AI102[2];//	正极倒角深度后纠偏检测
arrFilter_AD[8].AD	:=	AI102[3];//	备用

arrFilter_AD[9].AD		;//	正极
arrFilter_AD[10].AD		;//	正极
arrFilter_AD[11].AD		;//	正极
arrFilter_AD[12].AD		;//	正极

//负极
arrFilter_AD[13].AD	:=	AI201[0];//	负极左放卷卷径超声波检测
arrFilter_AD[14].AD	:=	AI201[1];//	负极右放卷卷径超声波检测
//arrFilter_AD[15].AD	:=	AI201[2];//	负极辅驱前料带张力检测
 arrFilter_ADV2[2].AD	:=	AI201[2];//	负极辅驱前料带张力检测
 
arrFilter_AD[16].AD	:=	AI201[3];//	备用
arrFilter_AD[17].AD	:=	AI202[0];//	负极后摆杆电位计检测
arrFilter_AD[18].AD	:=	AI202[1];//	负极倒角深度前纠偏检测
arrFilter_AD[19].AD	:=	AI202[2];//	负极倒角深度后纠偏检测
arrFilter_AD[20].AD	:=	AI202[3];//	备用

arrFilter_AD[21].AD		;//	负极
arrFilter_AD[22].AD		;//	负极
arrFilter_AD[23].AD		;//	负极
arrFilter_AD[24].AD		;//	负极

//转换
FOR  I1:=1 TO MaxAINo   DO
(*	
     arrFilter_AD[I1].fPointNum:=10;
	IF  I1=6 OR I1=7  OR  I1=18 OR I1=19  THEN         
         arrFilter_AD[I1].fPointNum:=20;
	END_IF	 
		 
   IF I1=3 OR I1=15  THEN
	    arrFilter_ADV2[I1].fPointNum:=1500;
	END_IF	
	*)
	IF  I1=6 OR I1=7  OR  I1=18 OR I1=19  THEN         
         arrFilter_AD[I1].fPointNum:=20;
   ELSIF I1=3 OR I1=15  THEN
	    arrFilter_ADV2[1].fPointNum:=1000;
		arrFilter_ADV2[2].fPointNum:=1000;
   ELSE
	   arrFilter_AD[I1].fPointNum:=10;
   END_IF

   IF I1=3   THEN
		   //arrFilter_AD[3].AD	:=	AI101[2];//	正极辅驱前料带张力检测
	   arrFilter_ADV2[1](   
		  iMode:=         2, 
		  AD:=               , 
		  iLimitH:=         ProductPar.parFilterAD[3].iLimitH  , 
		  iLimitL:=          ProductPar.parFilterAD[3].iLimitL   , 
		  fRangeH:=      ProductPar.parFilterAD[3].fRangeH , 
		  fRangeL:=       ProductPar.parFilterAD[3].fRangeL , 
		  fPointNum:=    , 
		  Out_Value=>   ProductPar.parFilterAD[3].Out_Value  );
		  
		//arrFilter_AD[15].AD	:=	AI201[2];//	负极辅驱前料带张力检测
	ELSIF I1=15   THEN
	  arrFilter_ADV2[2](   
		  iMode:=         2, 
		  AD:=               , 
		  iLimitH:=         ProductPar.parFilterAD[15].iLimitH  , 
		  iLimitL:=          ProductPar.parFilterAD[15].iLimitL   , 
		  fRangeH:=      ProductPar.parFilterAD[15].fRangeH , 
		  fRangeL:=       ProductPar.parFilterAD[15].fRangeL , 
		  fPointNum:=    , 
		  Out_Value=>   ProductPar.parFilterAD[15].Out_Value  );	
   ELSE
	  arrFilter_AD[I1](
		  iMode:=         2, 
		  AD:=               , 
		  iLimitH:=         ProductPar.parFilterAD[I1].iLimitH  , 
		  iLimitL:=          ProductPar.parFilterAD[I1].iLimitL   , 
		  fRangeH:=      ProductPar.parFilterAD[I1].fRangeH , 
		  fRangeL:=       ProductPar.parFilterAD[I1].fRangeL , 
		  fPointNum:=    , 
		  Out_Value=>   ProductPar.parFilterAD[I1].Out_Value  );
   END_IF	  
	  
END_FOR

  
	  
	  
	  


////////////////引用///////////////////////////
stAnUwindTen.fWindDiameter:=ProductPar.parFilterAD[1].Out_Value	;	//	正极左放卷卷径超声波检测
stAnUwindTen.fWindDiameter:=ProductPar.parFilterAD[2].Out_Value		;	//	正极右放卷卷径超声波检测
AnSenser.aiPoleTensionFr:=ProductPar.parFilterAD[3].Out_Value		;	//	正极辅驱前料带张力检测
ProductPar.parFilterAD[4].Out_Value	;	//	备用

stAnAuxDriverTen.fDanserDegree:=ProductPar.parFilterAD[5].Out_Value	;	//	正极后摆杆电位计检测
AnSenser.aiMouldRectifyFr:=ProductPar.parFilterAD[6].Out_Value	;	//	正极倒角深度前纠偏检测
AnSenser.aiMouldRectifyBe:=ProductPar.parFilterAD[7].Out_Value	;	//	正极倒角深度后纠偏检测
ProductPar.parFilterAD[8].Out_Value	;	//	备用

ProductPar.parFilterAD[9].Out_Value	;	//	正极
ProductPar.parFilterAD[10].Out_Value	;	//	正极
ProductPar.parFilterAD[11].Out_Value	;	//	正极
ProductPar.parFilterAD[12].Out_Value	;	//	正极

stCaUwindTen.fWindDiameter:=ProductPar.parFilterAD[13].Out_Value	;	//	负极左放卷卷径超声波检测
stCaUwindTen.fWindDiameter:=ProductPar.parFilterAD[14].Out_Value	;	//	负极右放卷卷径超声波检测
CaSenser.aiPoleTensionFr:=ProductPar.parFilterAD[15].Out_Value	;	//	负极辅驱前料带张力检测
ProductPar.parFilterAD[16].Out_Value	;	//	备用

stCaAuxDriverTen.fDanserDegree:=ProductPar.parFilterAD[17].Out_Value	;	//	负极后摆杆电位计检测
CaSenser.aiMouldRectifyFr:=ProductPar.parFilterAD[18].Out_Value		;	//	负极倒角深度前纠偏检测
CaSenser.aiMouldRectifyBe:=ProductPar.parFilterAD[19].Out_Value		;	//	负极倒角深度后纠偏检测
ProductPar.parFilterAD[20].Out_Value	;	//	备用

ProductPar.parFilterAD[21].Out_Value	;	//	负极	
ProductPar.parFilterAD[22].Out_Value	;	//	负极		
ProductPar.parFilterAD[23].Out_Value	;	//	负极		
ProductPar.parFilterAD[24].Out_Value	;	//	负极		





(*
//正极
arrFilter_AD[1].AD	:=	AI101[0];//	正极左放卷卷径超声波检测
arrFilter_AD[2].AD	:=	AI101[1];//	正极右放卷卷径超声波检测
arrFilter_AD[3].AD	:=	AI101[2];//	正极辅驱前料带张力检测
arrFilter_AD[4].AD	:=	AI101[3];//	备用
			
arrFilter_AD[5].AD	:=	AI102[0];//	正极后摆杆电位计检测
arrFilter_AD[6].AD	:=	AI102[1];//	正极倒角深度前纠偏检测
arrFilter_AD[7].AD	:=	AI102[2];//	正极倒角深度后纠偏检测
arrFilter_AD[8].AD	:=	AI102[3];//	备用

arrFilter_AD[9].AD		;//	正极
arrFilter_AD[10].AD		;//	正极
arrFilter_AD[11].AD		;//	正极
arrFilter_AD[12].AD		;//	正极

//负极
arrFilter_AD[13].AD	:=	AI201[0];//	负极左放卷卷径超声波检测
arrFilter_AD[14].AD	:=	AI201[1];//	负极右放卷卷径超声波检测
arrFilter_AD[15].AD	:=	AI201[2];//	负极辅驱前料带张力检测
arrFilter_AD[16].AD	:=	AI201[3];//	备用
			
arrFilter_AD[17].AD	:=	AI202[0];//	负极后摆杆电位计检测
arrFilter_AD[18].AD	:=	AI202[1];//	负极倒角深度前纠偏检测
arrFilter_AD[19].AD	:=	AI202[2];//	负极倒角深度后纠偏检测
arrFilter_AD[20].AD	:=	AI202[3];//	备用

arrFilter_AD[21].AD		;//	负极
arrFilter_AD[22].AD		;//	负极
arrFilter_AD[23].AD		;//	负极
arrFilter_AD[24].AD		;//	负极

//转换
FOR  I1:=1 TO MaxAINo   DO
	
	IF  I1=6 OR I1=7  OR  I1=18 OR I1=19  THEN         
         arrFilter_AD[I1].fPointNum:=40;
   ELSE
	   arrFilter_AD[I1].fPointNum:=10;
   END_IF
	
  arrFilter_AD[I1](
	  iMode:=         2, 
	  AD:=               , 
	  iLimitH:=         ProductPar.parFilterAD[I1].iLimitH  , 
	  iLimitL:=          ProductPar.parFilterAD[I1].iLimitL   , 
	  fRangeH:=      ProductPar.parFilterAD[I1].fRangeH , 
	  fRangeL:=       ProductPar.parFilterAD[I1].fRangeL , 
	  fPointNum:=    , 
	  Out_Value=>   ProductPar.parFilterAD[I1].Out_Value  );
END_FOR
////////////////引用///////////////////////////
stAnUwindTen.fWindDiameter:=ProductPar.parFilterAD[1].Out_Value	;	//	正极左放卷卷径超声波检测
stAnUwindTen.fWindDiameter:=ProductPar.parFilterAD[2].Out_Value		;	//	正极右放卷卷径超声波检测
AnSenser.aiPoleTensionFr:=ProductPar.parFilterAD[3].Out_Value		;	//	正极辅驱前料带张力检测
ProductPar.parFilterAD[4].Out_Value	;	//	备用

stAnAuxDriverTen.fDanserDegree:=ProductPar.parFilterAD[5].Out_Value	;	//	正极后摆杆电位计检测
AnSenser.aiMouldRectifyFr:=ProductPar.parFilterAD[6].Out_Value	;	//	正极倒角深度前纠偏检测
AnSenser.aiMouldRectifyBe:=ProductPar.parFilterAD[7].Out_Value	;	//	正极倒角深度后纠偏检测
ProductPar.parFilterAD[8].Out_Value	;	//	备用

ProductPar.parFilterAD[9].Out_Value	;	//	正极
ProductPar.parFilterAD[10].Out_Value	;	//	正极
ProductPar.parFilterAD[11].Out_Value	;	//	正极
ProductPar.parFilterAD[12].Out_Value	;	//	正极

stCaUwindTen.fWindDiameter:=ProductPar.parFilterAD[13].Out_Value	;	//	负极左放卷卷径超声波检测
stCaUwindTen.fWindDiameter:=ProductPar.parFilterAD[14].Out_Value	;	//	负极右放卷卷径超声波检测
CaSenser.aiPoleTensionFr:=ProductPar.parFilterAD[15].Out_Value	;	//	负极辅驱前料带张力检测
ProductPar.parFilterAD[16].Out_Value	;	//	备用

stCaAuxDriverTen.fDanserDegree:=ProductPar.parFilterAD[17].Out_Value	;	//	负极后摆杆电位计检测
CaSenser.aiMouldRectifyFr:=ProductPar.parFilterAD[18].Out_Value		;	//	负极倒角深度前纠偏检测
CaSenser.aiMouldRectifyBe:=ProductPar.parFilterAD[19].Out_Value		;	//	负极倒角深度后纠偏检测
ProductPar.parFilterAD[20].Out_Value	;	//	备用

ProductPar.parFilterAD[21].Out_Value	;	//	负极	
ProductPar.parFilterAD[22].Out_Value	;	//	负极		
ProductPar.parFilterAD[23].Out_Value	;	//	负极		
ProductPar.parFilterAD[24].Out_Value	;	//	负极		
*)
END_ACTION

ACTION AO:
////////模切AO部分////////				
AO101[0]:=REAL_TO_INT(ProductPar.parDA[1]*0.1+parDAOld[1]*0.9)			;	//	正极后摆杆比例阀
AO101[1]:=REAL_TO_INT(ProductPar.parDA[2]*0.1+parDAOld[2]*0.9)			;	//	正极主驱压辊比例阀
AO101[2]:=REAL_TO_INT(ProductPar.parDA[3]*0.1+parDAOld[3]*0.9)			;	//	正极
AO101[3]:=REAL_TO_INT(ProductPar.parDA[4]*0.1+parDAOld[4]*0.9)			;	//	正极
		
parDAOld[1]:=AO101[0];
parDAOld[2]:=AO101[1];
parDAOld[3]:=AO101[2];
parDAOld[4]:=AO101[3];
				
AO201[0]:=REAL_TO_INT(ProductPar.parDA[5]*0.1+parDAOld[5]*0.9)			;	//	负极后摆杆比例阀
AO201[1]:=REAL_TO_INT(ProductPar.parDA[6]*0.1+parDAOld[6]*0.9)			;	//	负极主驱压辊比例阀
AO201[2]:=REAL_TO_INT(ProductPar.parDA[7]*0.1+parDAOld[7]*0.9)			;	//	负极
AO201[3]:=REAL_TO_INT(ProductPar.parDA[8]*0.1+parDAOld[8]*0.9)			;	//	负极

parDAOld[5]:=AO201[0];
parDAOld[6]:=AO201[1];
parDAOld[7]:=AO201[2];
parDAOld[8]:=AO201[3];





///////////////正极张力转换///////////////////////////////
ProductPar.parFilterDA[1].bMode;  //TRUE 为标定模式      标定完成后一定要复位      

ProductPar.parFilterDA[1].X0;   //料带张力低限值    g
ProductPar.parFilterDA[1].Y0;    //料带张力低限值 DA输出   
ProductPar.parFilterDA[1].X1;  //料带张力高限值    g
ProductPar.parFilterDA[1].Y1;   //料带张力高限值   DA输出 
ProductPar.parFilterDA[1].iDAValue;   //标定DA值     

ProductPar.parDA[1]:=REAL_TO_INT(FC_Filter_AA(ProductPar.AnPar.fFr_TenValuehmi,0,0,100,30000));//	正极后摆杆比例阀
(*
ProductPar.parDA[1]:= SEL(ProductPar.parFilterDA[1].bMode,    
                                 REAL_TO_INT(FC_Filter_AA(ProductPar.AnPar.fFr_TenValuehmi,ProductPar.parFilterDA[1].X0,ProductPar.parFilterDA[1].Y0,ProductPar.parFilterDA[1].X1,ProductPar.parFilterDA[1].Y1)  ) ,     
                                 REAL_TO_INT (ProductPar.parFilterDA[1].iDAValue)   );                 //               REAL_TO_INT(FC_Filter_AA(ProductPar.AnPar.fFr_TenValuehmi,0,0,100,30000));//	正极后摆杆比例阀
*)
								 
ProductPar.parDA[2]:=REAL_TO_INT(FC_Filter_AA(ProductPar.AnPar.fPressDDRhmi,0,0,100,2000));//	正极主驱压辊比例阀
//AnPar.fBe_TenValue:=FC_Filter_AA(AnPar.fBe_TenValuehmi,0,0,100,100);//	正极前摆杆扭矩设置

///////////////负极张力转换///////////////////////////////
ProductPar.parFilterDA[2].bMode;  //TRUE 为标定模式      标定完成后一定要复位      

ProductPar.parFilterDA[2].X0;   //料带张力低限值    g
ProductPar.parFilterDA[2].Y0;    //料带张力低限值 DA输出   
ProductPar.parFilterDA[2].X1;  //料带张力高限值    g
ProductPar.parFilterDA[2].Y1;   //料带张力高限值   DA输出 
ProductPar.parFilterDA[2].iDAValue;   //标定DA值     
   
ProductPar.parDA[5]:=REAL_TO_INT(FC_Filter_AA(ProductPar.CaPar.fFr_TenValuehmi,0,0,100,30000));//	负极后摆杆比例阀
(*
ProductPar.parDA[5]:= SEL(ProductPar.parFilterDA[2].bMode,    
                                 REAL_TO_INT(FC_Filter_AA(ProductPar.CaPar.fFr_TenValuehmi,ProductPar.parFilterDA[2].X0,ProductPar.parFilterDA[2].Y0,ProductPar.parFilterDA[2].X1,ProductPar.parFilterDA[2].Y1)  ) ,     
                                  REAL_TO_INT(ProductPar.parFilterDA[2].iDAValue)  ) ;  
*)								  
								  
ProductPar.parDA[6]:=REAL_TO_INT(FC_Filter_AA(ProductPar.CaPar.fPressDDRhmi,0,0,100,2000));//	负极主驱压辊比例阀
//CaPar.fBe_TenValue:=FC_Filter_AA(CaPar.fBe_TenValuehmi,0,0,100,100);//	负极前摆杆扭矩设置
END_ACTION

ACTION InPut:


//输入映射	正极
		arrCyCtrl[NameNo.AnCYNo.BoardPressL].Io.DIONSwitch:=	I101[1]	;//	正极极片左接带气缸伸出位		
		arrCyCtrl[NameNo.AnCYNo.BoardPressL].Io.DIOFFSwitch:=	I101[2]	;//	正极极片左接带气缸缩回位		
		arrCyCtrl[NameNo.AnCYNo.BoardPressR].Io.DIONSwitch:=	I101[3]	;//	正极极片右接带气缸伸出位		
		arrCyCtrl[NameNo.AnCYNo.BoardPressR].Io.DIOFFSwitch:=	I101[4]	;//	正极极片右接带气缸缩回位		
		AnBtn.PoleBoxBit1:=	I101[5]	;//	正极放卷按钮BIT1		
		AnBtn.PoleBoxBit2:=	I101[6]	;//	正极放卷按钮BIT2		
		AnBtn.PoleBoxBit3:=	I101[7]	;//	正极放卷按钮BIT3		
		AnBtn.PoleBoxBit4:=	I101[8]	;//	正极放卷按钮BIT4		
		AnBtn.PoleBoxStart:=	I101[9]	;//	正极放卷启动按钮		
		AnBtn.PoleBoxEStop:=	I101[10]	;//	正极片放卷急停		
		AnBtn.CoderRollPress:=	I101[11]	;//	正极编码器压辊按钮		
			I101[12]	;//			
		arrCyCtrl[NameNo.AnCYNo.DriverPressAux].Io.DIONSwitch:=arrCyCtrl[NameNo.AnCYNo.DriverPressAux].Io.DOStatus1	;//I101[13]	;//	正极辅助驱动压辊伸出位		
		arrCyCtrl[NameNo.AnCYNo.DriverPressAux].Io.DIOFFSwitch:=NOT arrCyCtrl[NameNo.AnCYNo.DriverPressAux].Io.DOStatus1	;//I101[14]	;//	正极辅助驱动压辊缩回位		
		arrCyCtrl[NameNo.AnCYNo.CoderRollPress].Io.DIONSwitch:=	arrCyCtrl[NameNo.AnCYNo.CoderRollPress].Io.DOStatus1;//I101[15]	;//	正极前线扫编码器压辊伸出位		
		arrCyCtrl[NameNo.AnCYNo.CoderRollPress].Io.DIOFFSwitch:=	NOT arrCyCtrl[NameNo.AnCYNo.CoderRollPress].Io.DOStatus1;//I101[16]	;//	正极前线扫编码器压辊缩回位		
							
		AnBtn.DriverPress_Aux:=	I102[1]	;//	正极辅驱压辊旋钮		
		AnBtn.DriverJogFw_Aux:=	I102[2]	;//	正极辅驱正转旋钮		
		AnBtn.DriverJogBw_Aux:=	I102[3]	;//	正极辅驱反转旋钮		
			I102[4]	;//			
		arrRecCtrl[NameNo.AnRecNo.PoleWind].Io.biAutoDone:=	I102[5]	;//	正极放卷纠偏自动模式		
		arrRecCtrl[NameNo.AnRecNo.PoleWind].Io.biAlarm:=	I102[6]	;//	正极放卷纠偏故障		
		arrRecCtrl[NameNo.AnRecNo.PoleProcess].Io.biAutoDone:=	I102[7]	;//	正极行进纠偏自动模式		
		arrRecCtrl[NameNo.AnRecNo.PoleProcess].Io.biAlarm:=	I102[8]	;//	正极行进纠偏故障
			I102[9]	;//			
		AnSenser.biFlgBlue:=	I102[10]	;//	正极放卷蓝胶检测		
			AnSenser.bLineScanResult1_UP:=I102[11]	;//	正极CCD上线扫结果OK
			AnSenser.bLineScanResult2_UP:=I102[12]	;//	正极CCD上线扫结果NG		
			I102[13]	;//	
			AnSenser.bLineScanResult1_Down:=I102[14]	;//	正极CCD下线扫结果OK
			AnSenser.bLineScanResult2_Down:=I102[15]	;//	正极CCD下线扫结果NG
		//AnSenser.biTabHave:=	I102[16]	;//		极耳有无检测	
		AnSenser.bPoleCheck_R:=I102[16]	;//		正极倒角前极耳检测感应器					
		arrCyCtrl[NameNo.AnCYNo.DriverPressDDR].Io.DIONSwitch:=	I103[1]	;//	正极极主驱动压辊伸出位		
		arrCyCtrl[NameNo.AnCYNo.DriverPressDDR].Io.DIOFFSwitch:=	I103[2]	;//	正极极主驱动压辊缩回位		
		AnBtn.DriverPressDDR:=	I103[3]	;//	正极主驱动压辊按钮		
		AnSenser.biCuterStopUp:=	I103[4]	;//	正极裁切切刀堵料检测		
		AnSenser.biSafetyCurtain_M:=	I103[5]	;//	正极模具安全光栅		
		AnSenser.biSafetyCurtain_C:=	I103[6]	;//	正极裁切安全光栅		
		arrCyCtrl[NameNo.AnCYNo.NGRevBeltUpDown].Io.DIONSwitch:=	I103[7]	;//	正极踢废倒装皮带升降气缸伸出位		
		arrCyCtrl[NameNo.AnCYNo.NGRevBeltUpDown].Io.DIOFFSwitch:=	I103[8]	;//	正极踢废倒装皮带升降气缸缩回位		
		AnSenser.biWasteBox:=	I103[9]	;//	正极连续废料收集箱高度感应		
			I103[10]	;//			
		//arrCyCtrl[NameNo.AnCYNo.NGBoxLock1].Io.DIONSwitch:=	I103[11]	;//	正极NG收料归正伸出位1		
		//arrCyCtrl[NameNo.AnCYNo.NGBoxLock2].Io.DIONSwitch:=	I103[12]	;//	正极NG收料归正伸出位2		
		//arrCyCtrl[NameNo.AnCYNo.NGBoxLock1].Io.DIOFFSwitch:=	I103[13]	;//	正极NG收料归正缩回位1		
		//arrCyCtrl[NameNo.AnCYNo.NGBoxLock2].Io.DIOFFSwitch:=	I103[14]	;//	正极NG收料归正缩回位2		
		//AnBtn.NGBoxEStop:=//	I103[15]	;//	正极NG收料盒急停按钮		
		AnBtn.NGBoxStart:=	I103[16]	;//	正极NG收料盒确认放入料框按钮		
							
		AnBtn.NGBoxMotor_JogUp:=	I104[1]	;//	正极NG收料盒电机上升按钮		
		AnBtn.NGBoxMotor_JogDown:=	I104[2]	;//	正极NG收料盒电机下降按钮		
		AnsetpMotor.biSensor:=	I104[3]	;//	正极NG料盒高度感应		
		AnsetpMotor.biBoxSensor:=	I104[4]	;//	正极NG料盒到位感应		
		AnsetpMotor.biUpSensor:=	I104[5]	;//	正极NG料盒顶升电机上限		
		AnsetpMotor.biDownSensor:=	I104[6]	;//	正极NG料盒顶升电机下限		
		AnBtn.PoleBrushDustPush_U:=	I104[7]	;//	正极上表面毛刷除尘升降气缸按钮		
		AnBtn.PoleWindDustPush_U:=	I104[8]	;//	正极上表面超声波除尘升降气缸按钮		
		arrCyCtrl[NameNo.AnCYNo.PoleBrushDustPush_U].Io.DIONSwitch:=	I104[9]	;//	正极上表面毛刷除尘升降气缸伸出位		
		arrCyCtrl[NameNo.AnCYNo.PoleBrushDustPush_U].Io.DIOFFSwitch:=	I104[10]	;//	正极上表面毛刷除尘升降气缸缩回位		
		arrCyCtrl[NameNo.AnCYNo.PoleWindDustPush_U].Io.DIONSwitch:=	I104[11]	;//	正极上表面风刀除尘升降气缸伸出位		
		arrCyCtrl[NameNo.AnCYNo.PoleWindDustPush_U].Io.DIOFFSwitch:=	I104[12]	;//	正极上表面风刀除尘升降气缸缩回位		
		AnBtn.PoleBrushDustPush_D:=	I104[13]	;//	正极下表面毛刷除尘升降气缸按钮		
		AnBtn.PoleWindDustPush_D:=	I104[14]	;//	正极下表面超声波除尘升降气缸按钮		
		arrCyCtrl[NameNo.AnCYNo.DustRevBeltUpDown].Io.DIONSwitch:=	I104[15]	;//	正极下表面除尘倒装皮带升降气缸伸出位		
		arrCyCtrl[NameNo.AnCYNo.DustRevBeltUpDown].Io.DIOFFSwitch:=	I104[16]	;//	正极下表面除尘倒装皮带升降气缸缩回位		
							
		arrCyCtrl[NameNo.AnCYNo.PoleBrushDustPush_D].Io.DIONSwitch:=	I105[1]	;//	正极下表面毛刷除尘升降气缸伸出位		
		arrCyCtrl[NameNo.AnCYNo.PoleBrushDustPush_D].Io.DIOFFSwitch:=I105[2]	;//	正极下表面毛刷除尘升降气缸缩回位		
		arrCyCtrl[NameNo.AnCYNo.PoleWindDustPush_D].Io.DIONSwitch:=	I105[3]	;//	正极下表面风刀除尘升降气缸伸出位		
		arrCyCtrl[NameNo.AnCYNo.PoleWindDustPush_D].Io.DIOFFSwitch:=	I105[4]	;//	正极下表面风刀除尘升降气缸缩回位		
			I105[5]	;//			
		AnSenser.NGBoxFull:=I105[6]	;//正极NG料盒料满报警			
		AnSenser.NGboxsensor:=I105[7]	;//正极NG料盒抛料对射感应		
		AnSenser.bFourYellowDown:=I105[8]	;//	正极四连标下		
		AnSenser.bFourYellowUP:=I105[9]	;//	正极四连标上		
			I105[10]	;//			
			I105[11]	;//			
			I105[12]	;//			
			I105[13]	;//			
			I105[14]	;//			
			I105[15]	;//			
			I105[16]	;//			
							
		AnSys.btnAuto:=	I106[1]	;//	正极控制面板手自动切换按钮		
		AnSys.btnStart:=	I106[2]	;//	正极控制面板启动按钮		
		AnSys.btnReset:=	I106[3]	;//	正极控制面板复位按钮		
		AnSys.btnStop:=	I106[4]	;//	正极控制面板停止按钮		
		AnSys.btnEstop:=	I106[5]	AND I106[9];//	正极控制面板急停按钮		
		AnBtn.EncloserEstop[1]:=	I106[6]	;//	正极外罩急停1		
		AnBtn.EncloserEstop[2]:=	I106[7]	;//	正极外罩急停2		
		AnBtn.EncloserEstop[3]:=	I106[8]	;//	正极外罩急停3		
			//I106[9]	;//			
		AnSenser.biDoor[1]:=	I106[10]	;//	正极外罩门禁1		
		AnSenser.biDoor[2]:=	I106[11]	;//	正极外罩门禁2		
		AnSenser.biDoor[3]:=	I106[12]	;//	正极外罩门禁3		
		AnSenser.biDoor[4]:=	I106[13]	;//	正极外罩门禁4		
		AnSenser.biDoor[5]:=	I106[14]	;//	正极外罩门禁5		
			I106[15]	;//		
			I106[16]	;//		
							
			I107[1]	;//			
			I107[2]	;//			
			I107[3]	;//			
			I107[4]	;//			
			I107[5]	;//			
			I107[6]	;//			
			I107[7]	;//			
			I107[8]	;//			
			I107[9]	;//			
			I107[10]	;//			
			I107[11]	;//			
			I107[12]	;//			
			I107[13]	;//			
			I107[14]	;//			
			I107[15]	;//			
			I107[16]	;//			
			AnSenser.aThrow:=	I104[9]	;//	正极上表面毛刷除尘升降气缸伸出位(踢废失败报警解除专用)	
			AnSenser.biCutPoleHave	:=	I108[1]	;	//裁切后极片有无检测	
			AnSenser.bKick :=I108[2]	;//	踢废工位有无料检测；		
			AnSenser.bYellowCheck_C:=I108[3]	;//	正极踢废前黄标检测感应器；		
			AnSenser.bYellowCheck_R1:=I108[4]	;//正极倒角前接带检测感应器	上	
			//AnSenser.bPoleCheck_R:=I108[5]	;//		正极倒角前极耳检测感应器
			AnSenser.bYellowCheck_R2:=I108[6]	;//	正极倒角前接带检测感应器下
			AnSenser.MouldInsensor:=I108[7]	;//	//R角模具到位感应		
			AnSenser.CuterInsensor:=I108[8]	;//裁切切刀到位感应		
			I108[9]	;//			
			I108[10]	;//			
			I108[11]	;//			
			I108[12]	;//			
			I108[13]	;//			
			I108[14]	;//			
			I108[15]	;//			
			I108[16]	;//			
							
			I109[1]	;//			
			I109[2]	;//			
			I109[3]	;//			
			I109[4]	;//			
			I109[5]	;//			
			I109[6]	;//			
			I109[7]	;//			
			I109[8]	;//			
			I109[9]	;//			
			I109[10]	;//			
			I109[11]	;//			
			I109[12]	;//			
			I109[13]	;//			
			I109[14]	;//			
			I109[15]	;//			
			I109[16]	;//			
			
			AnSenser.biSubBelt1Have:=I30101;	//	1号叠台:正极模切送料分段皮带1有料感应
			AnSenser.biSubBelt2Have:=I40101;	//	2号叠台:正极模切送料分段皮带2有料感应	
			AnSenser.biSubBelt3Have:=I50101;	//	3号叠台:正极模切送料分段皮带3有料感应		
//输入映射	负极						
		arrCyCtrl[NameNo.CaCYNo.BoardPressL].Io.DIONSwitch:=	I201[1]	;//	负极极片左接带气缸伸出位		
		arrCyCtrl[NameNo.CaCYNo.BoardPressL].Io.DIOFFSwitch:=	I201[2]	;//	负极极片左接带气缸缩回位		
		arrCyCtrl[NameNo.CaCYNo.BoardPressR].Io.DIONSwitch:=	I201[3]	;//	负极极片右接带气缸伸出位		
		arrCyCtrl[NameNo.CaCYNo.BoardPressR].Io.DIOFFSwitch:=	I201[4]	;//	负极极片右接带气缸缩回位		
		CaBtn.PoleBoxBit1:=	I201[5]	;//	负极放卷按钮BIT1		
		CaBtn.PoleBoxBit2:=	I201[6]	;//	负极放卷按钮BIT2		
		CaBtn.PoleBoxBit3:=	I201[7]	;//	负极放卷按钮BIT3		
		CaBtn.PoleBoxBit4:=	I201[8]	;//	负极放卷按钮BIT4		
		CaBtn.PoleBoxStart:=	I201[9]	;//	负极放卷启动按钮		
		CaBtn.PoleBoxEStop:=	I201[10]	;//	负极片放卷急停		
		CaBtn.CoderRollPress:=	I201[11]	;//	负极编码器压辊按钮
			I201[12]	;//			
		arrCyCtrl[NameNo.CaCYNo.DriverPressAux].Io.DIONSwitch:=arrCyCtrl[NameNo.CaCYNo.DriverPressAux].Io.DOStatus1	;//I201[13]	;//	负极辅助驱动压辊伸出位		
		arrCyCtrl[NameNo.CaCYNo.DriverPressAux].Io.DIOFFSwitch:=NOT arrCyCtrl[NameNo.CaCYNo.DriverPressAux].Io.DOStatus1	;//I201[14]	;//	负极辅助驱动压辊缩回位		
		arrCyCtrl[NameNo.CaCYNo.CoderRollPress].Io.DIONSwitch:=arrCyCtrl[NameNo.CaCYNo.CoderRollPress].Io.DOStatus1	;//I201[15]	;//	负极前线扫编码器压辊伸出位		
		arrCyCtrl[NameNo.CaCYNo.CoderRollPress].Io.DIOFFSwitch:=NOT arrCyCtrl[NameNo.CaCYNo.CoderRollPress].Io.DOStatus1	;//I201[16]	;//	负极前线扫编码器压辊缩回位		
							
		CaBtn.DriverPress_Aux:=	I202[1]	;//	负极辅驱压辊旋钮		
		CaBtn.DriverJogFw_Aux:=	I202[2]	;//	负极辅驱正转旋钮		
		CaBtn.DriverJogBw_Aux:=	I202[3]	;//	负极辅驱反转旋钮		
			I202[4]	;//			
		arrRecCtrl[NameNo.CaRecNo.PoleWind].Io.biAutoDone:=	I202[5]	;//	负极放卷纠偏自动模式		
		arrRecCtrl[NameNo.CaRecNo.PoleWind].Io.biAlarm:=	I202[6]	;//	负极放卷纠偏故障	
		arrRecCtrl[NameNo.CaRecNo.PoleProcess].Io.biAutoDone:=	I202[7]	;//	负极行进纠偏自动模式		
		arrRecCtrl[NameNo.CaRecNo.PoleProcess].Io.biAlarm:=	I202[8]	;//	负极行进纠偏故障		
			I202[9]	;//			
		CaSenser.biFlgBlue:=	I202[10]	;//	负极放卷蓝胶检测	
			CaSenser.bLineScanResult1_UP:=I202[11]	;//	负极CCD上线扫结果OK
			CaSenser.bLineScanResult2_UP:=I202[12]	;//	负极CCD上线扫结果NG
			I202[13]	;//	
			CaSenser.bLineScanResult1_Down:=I202[14]	;//	负极CCD下线扫结果OK
			CaSenser.bLineScanResult2_Down:=I202[15]	;//	负极CCD下线扫结果NG
		//CaSenser.biTabHave:=	I202[16]	;//		极耳有无检测	
		CaSenser.bPoleCheck_R:=I202[16]	;//	负极倒角前极耳检测感应器					
		arrCyCtrl[NameNo.CaCYNo.DriverPressDDR].Io.DIONSwitch:=	I203[1]	;//	负极极主驱动压辊伸出位		
		arrCyCtrl[NameNo.CaCYNo.DriverPressDDR].Io.DIOFFSwitch:=	I203[2]	;//	负极极主驱动压辊缩回位		
		CaBtn.DriverPressDDR:=	I203[3]	;//	负极主驱动压辊按钮		
		CaSenser.biCuterStopUp:=	I203[4]	;//	负极裁切切刀堵料检测		
		CaSenser.biSafetyCurtain_M:=	I203[5]	;//	负极模具安全光栅		
		CaSenser.biSafetyCurtain_C:=	I203[6]	;//	负极裁切安全光栅		
		arrCyCtrl[NameNo.CaCYNo.NGRevBeltUpDown].Io.DIONSwitch:=	I203[7]	;//	负极踢废倒装皮带升降气缸伸出位		
		arrCyCtrl[NameNo.CaCYNo.NGRevBeltUpDown].Io.DIOFFSwitch:=	I203[8]	;//	负极踢废倒装皮带升降气缸缩回位		
		CaSenser.biWasteBox:=	I203[9]	;//	负极连续废料收集箱高度感应		
			I203[10]	;//			
		//arrCyCtrl[NameNo.CaCYNo.NGBoxLock1].Io.DIONSwitch:=	I203[11]	;//	负极NG收料归正伸出位1		
		//arrCyCtrl[NameNo.CaCYNo.NGBoxLock2].Io.DIONSwitch:=	I203[12]	;//	负极NG收料归正伸出位2		
		//arrCyCtrl[NameNo.CaCYNo.NGBoxLock1].Io.DIOFFSwitch:=	I203[13]	;//	负极NG收料归正缩回位1		
		//arrCyCtrl[NameNo.CaCYNo.NGBoxLock2].Io.DIOFFSwitch:=	I203[14]	;//	负极NG收料归正缩回位2		
		CaBtn.NGBoxEStop:=//	I203[15]	;//	负极NG收料盒急停按钮		
		CaBtn.NGBoxStart:=	I203[16]	;//	负极NG收料盒确认放入料框按钮		
							
		CaBtn.NGBoxMotor_JogUp:=	I204[1]	;//	负极NG收料盒电机上升按钮		
		CaBtn.NGBoxMotor_JogDown:=	I204[2]	;//	负极NG收料盒电机下降按钮		
		CasetpMotor.biSensor:=	I204[3]	;//	负极NG料盒高度感应		
		CasetpMotor.biBoxSensor:=	I204[4]	;//	负极NG料盒到位感应		
		CasetpMotor.biUpSensor:=	I204[5]	;//	负极NG料盒顶升电机上限		
		CasetpMotor.biDownSensor:=	I204[6]	;//	负极NG料盒顶升电机下限		
		CaBtn.PoleBrushDustPush_U:=	I204[7]	;//	负极上表面毛刷除尘升降气缸按钮		
		CaBtn.PoleWindDustPush_U:=	I204[8]	;//	负极上表面超声波除尘升降气缸按钮		
		arrCyCtrl[NameNo.CaCYNo.PoleBrushDustPush_U].Io.DIONSwitch:=	I204[9]	;//	负极上表面毛刷除尘升降气缸伸出位		
		arrCyCtrl[NameNo.CaCYNo.PoleBrushDustPush_U].Io.DIOFFSwitch:=	I204[10]	;//	负极上表面毛刷除尘升降气缸缩回位		
		arrCyCtrl[NameNo.CaCYNo.PoleWindDustPush_U].Io.DIONSwitch:=	I204[11]	;//	负极上表面风刀除尘升降气缸伸出位		
		arrCyCtrl[NameNo.CaCYNo.PoleWindDustPush_U].Io.DIOFFSwitch:=	I204[12]	;//	负极上表面风刀除尘升降气缸缩回位		
		CaBtn.PoleBrushDustPush_D:=	I204[13]	;//	负极下表面毛刷除尘升降气缸按钮		
		CaBtn.PoleWindDustPush_D:=	I204[14]	;//	负极下表面超声波除尘升降气缸按钮		
		arrCyCtrl[NameNo.CaCYNo.DustRevBeltUpDown].Io.DIONSwitch:=	I204[15]	;//	负极下表面除尘倒装皮带升降气缸伸出位		
		arrCyCtrl[NameNo.CaCYNo.DustRevBeltUpDown].Io.DIOFFSwitch:=	I204[16]	;//	负极下表面除尘倒装皮带升降气缸缩回位		
							
		arrCyCtrl[NameNo.CaCYNo.PoleBrushDustPush_D].Io.DIONSwitch:=	I205[1]	;//	负极下表面毛刷除尘升降气缸伸出位		
		arrCyCtrl[NameNo.CaCYNo.PoleBrushDustPush_D].Io.DIOFFSwitch:=	I205[2]	;//	负极下表面毛刷除尘升降气缸缩回位		
		arrCyCtrl[NameNo.CaCYNo.PoleWindDustPush_D].Io.DIONSwitch:=	I205[3]	;//	负极下表面风刀除尘升降气缸伸出位		
		arrCyCtrl[NameNo.CaCYNo.PoleWindDustPush_D].Io.DIOFFSwitch:=	I205[4]	;//	负极下表面风刀除尘升降气缸缩回位		
		I205[5]	;//	正压压力表；		
		CaSenser.NGBoxFull:=I205[6]	;//负极NG料盒料满报警			
		CaSenser.NGboxsensor :=I205[7]	;//负极NG料盒抛料对射感应		
		CaSenser.bFourYellowDown:=I205[8]	;//	负极四连标下		
		CaSenser.bFourYellowUP:=I205[9]	;//	负极四连标上		
			I205[10]	;//			
			I205[11]	;//			
			I205[12]	;//			
			I205[13]	;//			
			I205[14]	;//			
			I205[15]	;//			
			I205[16]	;//			
							
		CaSys.btnAuto:=	I206[1]	;//	负极控制面板手自动切换按钮		
		CaSys.btnStart:=	I206[2]	;//	负极控制面板启动按钮		
		CaSys.btnReset:=	I206[3]	;//	负极控制面板复位按钮		
		CaSys.btnStop:=	I206[4]	;//	负极控制面板停止按钮		
		CaSys.btnEstop:=	I206[5] AND I206[9]	;//	负极控制面板急停按钮		
		CaBtn.EncloserEstop[1]:=	I206[6]	;//	负极外罩急停1		
		CaBtn.EncloserEstop[2]:=	I206[7]	;//	负极外罩急停2		
		CaBtn.EncloserEstop[3]:=	I206[8]	;//	负极外罩急停3		
			//I206[9]	;//			
		CaSenser.biDoor[1]:=	I206[10]	;//	负极外罩门禁1		
		CaSenser.biDoor[2]:=	I206[11]	;//	负极外罩门禁2		
		CaSenser.biDoor[3]:=	I206[12]	;//	负极外罩门禁3		
		CaSenser.biDoor[4]:=	I206[13]	;//	负极外罩门禁4		
		CaSenser.biDoor[5]:=	I206[14]	;//	负极
			I206[15]	;//模切通道安全门报警
			I206[16]	;	
							
			I207[1]	;//			
			I207[2]	;//			
			I207[3]	;//			
			I207[4]	;//			
			I207[5]	;//			
			I207[6]	;//			
			I207[7]	;//			
			I207[8]	;//			
			I207[9]	;//			
			I207[10]	;//			
			I207[11]	;//			
			I207[12]	;//			
			I207[13]	;//			
			I207[14]	;//			
			I207[15]	;//			
			I207[16]	;//		
			CaSenser.aThrow:=	I204[9]	;//负极上表面毛刷除尘升降气缸伸出位(踢废失败报警解除专用)					
			CaSenser.biCutPoleHave	:=	I208[1]	;	//裁切后极片有无检测	
			CaSenser.bKick :=I208[2]	;//	踢废工位有无料检测；		
			CaSenser.bYellowCheck_C:=I208[3]	;//	负极色标传感器；		
			CaSenser.bYellowCheck_R1:=I208[4]	;//负极倒角前接带检测感应器上		
			//CaSenser.bPoleCheck_R:=I208[5]	;//	负极倒角前极耳检测感应器
			CaSenser.bYellowCheck_R2:=I208[6]	;//	负极倒角前接带检测感应器下
			CaSenser.MouldInsensor:=I208[7]	;//	R角模具到位感应		
			CaSenser.CuterInsensor:=I208[8]	;//	裁切切刀到位感应		
			I208[9]	;//			
			I208[10]	;//			
			I208[11]	;//			
			I208[12]	;//			
			I208[13]	;//			
			I208[14]	;//			
			I208[15]	;//			
			I208[16]	;//			
							
			I209[1]	;//			
			I209[2]	;//			
			I209[3]	;//			
			I209[4]	;//			
			I209[5]	;//			
			I209[6]	;//			
			I209[7]	;//			
			I209[8]	;//			
			I209[9]	;//			
			I209[10]	;//			
			I209[11]	;//			
			I209[12]	;//			
			I209[13]	;//			
			I209[14]	;//			
			I209[15]	;//			
			I209[16]	;//			

			CaSenser.biSubBelt1Have:=I30107;	//	1号叠台:负极模切送料分段皮带1有料感应
			CaSenser.biSubBelt2Have:=I40107;	//	2号叠台:负极模切送料分段皮带2有料感应	
			CaSenser.biSubBelt3Have:=I50107;	//	3号叠台:负极模切送料分段皮带3有料感应
END_ACTION

ACTION LimitSwitch:
//正极极片张力
arrAxisCtrl[NameNo.AnAxisNo.PoleTension].Io.DigitalInputs;
//arrAxisCtrl[NameNo.AnAxisNo.PoleTension].Io.biHomeSwitch:=arrAxisCtrl[NameNo.AnAxisNo.PoleTension].Io.DigitalInputs.2;
arrAxisCtrl[NameNo.AnAxisNo.PoleTension].Io.biNegLimit:=arrAxisCtrl[NameNo.AnAxisNo.PoleTension].Io.DigitalInputs.17;
arrAxisCtrl[NameNo.AnAxisNo.PoleTension].Io.biPosLimit:=arrAxisCtrl[NameNo.AnAxisNo.PoleTension].Io.DigitalInputs.16;
//arrAxisPar[NameNo.AnAxisNo.PoleTension].bLimitSwitchEn:=TRUE;//开启限位保护

//正极极片缓存
arrAxisCtrl[NameNo.AnAxisNo.BuffeLine].Io.DigitalInputs;
arrAxisCtrl[NameNo.AnAxisNo.BuffeLine].Io.biHomeSwitch:=arrAxisCtrl[NameNo.AnAxisNo.BuffeLine].Io.DigitalInputs.2;
arrAxisCtrl[NameNo.AnAxisNo.BuffeLine].Io.biNegLimit:= arrAxisCtrl[NameNo.AnAxisNo.BuffeLine].Io.DigitalInputs.17;
arrAxisCtrl[NameNo.AnAxisNo.BuffeLine].Io.biPosLimit:= arrAxisCtrl[NameNo.AnAxisNo.BuffeLine].Io.DigitalInputs.18;
arrAxisPar[NameNo.AnAxisNo.BuffeLine].bLimitSwitchEn:=TRUE;//开启限位保护

//正极模具纠偏X轴(肩宽)
arrAxisCtrl[NameNo.AnAxisNo.MouldRectify_X].Io.DigitalInputs;
arrAxisCtrl[NameNo.AnAxisNo.MouldRectify_X].Io.biHomeSwitch:=arrAxisCtrl[NameNo.AnAxisNo.MouldRectify_X].Io.DigitalInputs.2;
arrAxisCtrl[NameNo.AnAxisNo.MouldRectify_X].Io.biNegLimit:=arrAxisCtrl[NameNo.AnAxisNo.MouldRectify_X].Io.DigitalInputs.17;
arrAxisCtrl[NameNo.AnAxisNo.MouldRectify_X].Io.biPosLimit:=arrAxisCtrl[NameNo.AnAxisNo.MouldRectify_X].Io.DigitalInputs.16;
arrAxisPar[NameNo.AnAxisNo.MouldRectify_X].bLimitSwitchEn:=TRUE;//开启限位保护

//正极模具纠偏Y轴(切刀深度)   负限当作原点&负限
arrAxisCtrl[NameNo.AnAxisNo.MouldRectify_Y].Io.DigitalInputs;
arrAxisCtrl[NameNo.AnAxisNo.MouldRectify_Y].Io.biHomeSwitch:=arrAxisCtrl[NameNo.AnAxisNo.MouldRectify_Y].Io.DigitalInputs.17;
arrAxisCtrl[NameNo.AnAxisNo.MouldRectify_Y].Io.biNegLimit:=arrAxisCtrl[NameNo.AnAxisNo.MouldRectify_Y].Io.DigitalInputs.17;
arrAxisCtrl[NameNo.AnAxisNo.MouldRectify_Y].Io.biPosLimit:=arrAxisCtrl[NameNo.AnAxisNo.MouldRectify_Y].Io.DigitalInputs.16;
arrAxisPar[NameNo.AnAxisNo.MouldRectify_Y].bLimitSwitchEn:=TRUE;//开启限位保护

//正极模具
arrAxisCtrl[NameNo.AnAxisNo.Mould].Io.DigitalInputs;
arrAxisCtrl[NameNo.AnAxisNo.Mould].Io.biHomeSwitch:=arrAxisCtrl[NameNo.AnAxisNo.Mould].Io.DigitalInputs.2;
//arrAxisCtrl[AnAxisNo.Mould].Io.biNegLimit:=arrAxisCtrl[AnAxisNo.Mould].Io.DigitalInputs.0;
//arrAxisCtrl[AnAxisNo.Mould].Io.biPosLimit:=arrAxisCtrl[AnAxisNo.Mould].Io.DigitalInputs.1;

//正极裁切
arrAxisCtrl[NameNo.AnAxisNo.Cuter].Io.DigitalInputs;
arrAxisCtrl[NameNo.AnAxisNo.Cuter].Io.biHomeSwitch:=arrAxisCtrl[NameNo.AnAxisNo.Cuter].Io.DigitalInputs.2;
//arrAxisCtrl[AnAxisNo.Cuter].Io.biNegLimit:=arrAxisCtrl[AnAxisNo.Cuter].Io.DigitalInputs.0;
//arrAxisCtrl[AnAxisNo.Cuter].Io.biPosLimit:=arrAxisCtrl[AnAxisNo.Cuter].Io.DigitalInputs.1;

//正极裁切角度纠偏   负限当作原点&负限
arrAxisCtrl[NameNo.AnAxisNo.CuterDegRectify].Io.DigitalInputs;
arrAxisCtrl[NameNo.AnAxisNo.CuterDegRectify].Io.biHomeSwitch:=arrAxisCtrl[NameNo.AnAxisNo.CuterDegRectify].Io.DigitalInputs.17;
arrAxisCtrl[NameNo.AnAxisNo.CuterDegRectify].Io.biNegLimit:=arrAxisCtrl[NameNo.AnAxisNo.CuterDegRectify].Io.DigitalInputs.17;
arrAxisCtrl[NameNo.AnAxisNo.CuterDegRectify].Io.biPosLimit:=arrAxisCtrl[NameNo.AnAxisNo.CuterDegRectify].Io.DigitalInputs.16;
arrAxisPar[NameNo.AnAxisNo.CuterDegRectify].bLimitSwitchEn:=TRUE;//开启限位保护

//正极裁切换型
arrAxisCtrl[NameNo.AnAxisNo.CuterBeltChange].Io.DigitalInputs;
arrAxisCtrl[NameNo.AnAxisNo.CuterBeltChange].Io.biHomeSwitch:=arrAxisCtrl[NameNo.AnAxisNo.CuterBeltChange].Io.DigitalInputs.2;
arrAxisCtrl[NameNo.AnAxisNo.CuterBeltChange].Io.biNegLimit:=arrAxisCtrl[NameNo.AnAxisNo.CuterBeltChange].Io.DigitalInputs.17;
arrAxisCtrl[NameNo.AnAxisNo.CuterBeltChange].Io.biPosLimit:=arrAxisCtrl[NameNo.AnAxisNo.CuterBeltChange].Io.DigitalInputs.16;
arrAxisPar[NameNo.AnAxisNo.CuterBeltChange].bLimitSwitchEn:=TRUE;//开启限位保护

//正极初始踢废料
//arrAxisCtrl[NameNo.AnAxisNo.NGPush1].Io.DigitalInputs;
//arrAxisCtrl[NameNo.AnAxisNo.NGPush1].Io.biHomeSwitch:=NOT arrAxisCtrl[NameNo.AnAxisNo.NGPush1].Io.DigitalInputs.2;
//arrAxisCtrl[AnAxisNo.NGPush1].Io.biNegLimit:=arrAxisCtrl[AnAxisNo.NGPush1].Io.DigitalInputs.0;
//arrAxisCtrl[AnAxisNo.NGPush1].Io.biPosLimit:=arrAxisCtrl[AnAxisNo.NGPush1].Io.DigitalInputs.1;

//正极踢废料
//arrAxisCtrl[NameNo.AnAxisNo.NGPush2].Io.DigitalInputs;
//arrAxisCtrl[NameNo.AnAxisNo.NGPush2].Io.biHomeSwitch:=NOT arrAxisCtrl[NameNo.AnAxisNo.NGPush2].Io.DigitalInputs.2;
//arrAxisCtrl[AnAxisNo.NGPush2].Io.biNegLimit:=arrAxisCtrl[AnAxisNo.NGPush2].Io.DigitalInputs.0;
//arrAxisCtrl[AnAxisNo.NGPush2].Io.biPosLimit:=arrAxisCtrl[AnAxisNo.NGPush2].Io.DigitalInputs.1;

//正极CCD压片升降
arrAxisCtrl[NameNo.AnAxisNo.CCDPressPush].Io.DigitalInputs;
arrAxisCtrl[NameNo.AnAxisNo.CCDPressPush].Io.biHomeSwitch:=NOT arrAxisCtrl[NameNo.AnAxisNo.CCDPressPush].Io.DigitalInputs.2;
//arrAxisCtrl[AnAxisNo.CCDPressPush].Io.biNegLimit:=arrAxisCtrl[AnAxisNo.CCDPressPush].Io.DigitalInputs.0;
//arrAxisCtrl[AnAxisNo.CCDPressPush].Io.biPosLimit:=arrAxisCtrl[AnAxisNo.CCDPressPush].Io.DigitalInputs.1;


//负极极片张力
arrAxisCtrl[NameNo.CaAxisNo.PoleTension].Io.DigitalInputs;
//arrAxisCtrl[NameNo.CaAxisNo.PoleTension].Io.biHomeSwitch:=arrAxisCtrl[NameNo.CaAxisNo.PoleTension].Io.DigitalInputs.2;
arrAxisCtrl[NameNo.CaAxisNo.PoleTension].Io.biNegLimit:=arrAxisCtrl[NameNo.CaAxisNo.PoleTension].Io.DigitalInputs.17;
arrAxisCtrl[NameNo.CaAxisNo.PoleTension].Io.biPosLimit:=arrAxisCtrl[NameNo.CaAxisNo.PoleTension].Io.DigitalInputs.16;

//负极极片缓存
arrAxisCtrl[NameNo.CaAxisNo.BuffeLine].Io.DigitalInputs;
arrAxisCtrl[NameNo.CaAxisNo.BuffeLine].Io.biHomeSwitch:=arrAxisCtrl[NameNo.CaAxisNo.BuffeLine].Io.DigitalInputs.2;
arrAxisCtrl[NameNo.CaAxisNo.BuffeLine].Io.biNegLimit:= arrAxisCtrl[NameNo.CaAxisNo.BuffeLine].Io.DigitalInputs.17;
arrAxisCtrl[NameNo.CaAxisNo.BuffeLine].Io.biPosLimit:= arrAxisCtrl[NameNo.CaAxisNo.BuffeLine].Io.DigitalInputs.18;
arrAxisPar[NameNo.CaAxisNo.BuffeLine].bLimitSwitchEn:=TRUE;//开启限位保护

//负极模具纠偏X轴(肩宽)
arrAxisCtrl[NameNo.CaAxisNo.MouldRectify_X].Io.DigitalInputs;
arrAxisCtrl[NameNo.CaAxisNo.MouldRectify_X].Io.biHomeSwitch:=arrAxisCtrl[NameNo.CaAxisNo.MouldRectify_X].Io.DigitalInputs.2;
arrAxisCtrl[NameNo.CaAxisNo.MouldRectify_X].Io.biNegLimit:=arrAxisCtrl[NameNo.CaAxisNo.MouldRectify_X].Io.DigitalInputs.17;
arrAxisCtrl[NameNo.CaAxisNo.MouldRectify_X].Io.biPosLimit:=arrAxisCtrl[NameNo.CaAxisNo.MouldRectify_X].Io.DigitalInputs.16;
arrAxisPar[NameNo.CaAxisNo.MouldRectify_X].bLimitSwitchEn:=TRUE;//开启限位保护

//负极模具纠偏Y轴(切刀深度) 负限当作原点&负限
arrAxisCtrl[NameNo.CaAxisNo.MouldRectify_Y].Io.DigitalInputs;
arrAxisCtrl[NameNo.CaAxisNo.MouldRectify_Y].Io.biHomeSwitch:=arrAxisCtrl[NameNo.CaAxisNo.MouldRectify_Y].Io.DigitalInputs.17;//arrAxisCtrl[NameNo.CaAxisNo.MouldRectify_Y].Io.DigitalInputs.2;
arrAxisCtrl[NameNo.CaAxisNo.MouldRectify_Y].Io.biNegLimit:=arrAxisCtrl[NameNo.CaAxisNo.MouldRectify_Y].Io.DigitalInputs.17;
arrAxisCtrl[NameNo.CaAxisNo.MouldRectify_Y].Io.biPosLimit:=arrAxisCtrl[NameNo.CaAxisNo.MouldRectify_Y].Io.DigitalInputs.16;
arrAxisPar[NameNo.CaAxisNo.MouldRectify_Y].bLimitSwitchEn:=TRUE;//开启限位保护

//负极模具
arrAxisCtrl[NameNo.CaAxisNo.Mould].Io.DigitalInputs;
arrAxisCtrl[NameNo.CaAxisNo.Mould].Io.biHomeSwitch:=arrAxisCtrl[NameNo.CaAxisNo.Mould].Io.DigitalInputs.2;
//arrAxisCtrl[NameNo.CaAxisNo.Mould].Io.biNegLimit:=arrAxisCtrl[NameNo.CaAxisNo.Mould].Io.DigitalInputs.0;
//arrAxisCtrl[NameNo.CaAxisNo.Mould].Io.biPosLimit:=arrAxisCtrl[NameNo.CaAxisNo.Mould].Io.DigitalInputs.1;

//负极裁切
arrAxisCtrl[NameNo.CaAxisNo.Cuter].Io.DigitalInputs;
arrAxisCtrl[NameNo.CaAxisNo.Cuter].Io.biHomeSwitch:=arrAxisCtrl[NameNo.CaAxisNo.Cuter].Io.DigitalInputs.2;
//arrAxisCtrl[NameNo.CaAxisNo.Cuter].Io.biNegLimit:=arrAxisCtrl[NameNo.CaAxisNo.Cuter].Io.DigitalInputs.0;
//arrAxisCtrl[NameNo.CaAxisNo.Cuter].Io.biPosLimit:=arrAxisCtrl[NameNo.CaAxisNo.Cuter].Io.DigitalInputs.1;

//负极裁切角度纠偏   负限当作原点&负限
arrAxisCtrl[NameNo.CaAxisNo.CuterDegRectify].Io.DigitalInputs;
arrAxisCtrl[NameNo.CaAxisNo.CuterDegRectify].Io.biHomeSwitch:=arrAxisCtrl[NameNo.CaAxisNo.CuterDegRectify].Io.DigitalInputs.17;
arrAxisCtrl[NameNo.CaAxisNo.CuterDegRectify].Io.biNegLimit:=arrAxisCtrl[NameNo.CaAxisNo.CuterDegRectify].Io.DigitalInputs.17;
arrAxisCtrl[NameNo.CaAxisNo.CuterDegRectify].Io.biPosLimit:=arrAxisCtrl[NameNo.CaAxisNo.CuterDegRectify].Io.DigitalInputs.16;
arrAxisPar[NameNo.CaAxisNo.CuterDegRectify].bLimitSwitchEn:=TRUE;//开启限位保护

//负极裁切换型
arrAxisCtrl[NameNo.CaAxisNo.CuterBeltChange].Io.DigitalInputs;
arrAxisCtrl[NameNo.CaAxisNo.CuterBeltChange].Io.biHomeSwitch:=arrAxisCtrl[NameNo.CaAxisNo.CuterBeltChange].Io.DigitalInputs.2;
arrAxisCtrl[NameNo.CaAxisNo.CuterBeltChange].Io.biNegLimit:=arrAxisCtrl[NameNo.CaAxisNo.CuterBeltChange].Io.DigitalInputs.17;
arrAxisCtrl[NameNo.CaAxisNo.CuterBeltChange].Io.biPosLimit:=arrAxisCtrl[NameNo.CaAxisNo.CuterBeltChange].Io.DigitalInputs.16;
arrAxisPar[NameNo.CaAxisNo.CuterBeltChange].bLimitSwitchEn:=TRUE;//开启限位保护

//负极初始踢废料
//arrAxisCtrl[NameNo.CaAxisNo.NGPush1].Io.DigitalInputs;
//arrAxisCtrl[NameNo.CaAxisNo.NGPush1].Io.biHomeSwitch:=NOT arrAxisCtrl[NameNo.CaAxisNo.NGPush1].Io.DigitalInputs.2;
//arrAxisCtrl[NameNo.CaAxisNo.NGPush1].Io.biNegLimit:=arrAxisCtrl[NameNo.CaAxisNo.NGPush1].Io.DigitalInputs.0;
//arrAxisCtrl[NameNo.CaAxisNo.NGPush1].Io.biPosLimit:=arrAxisCtrl[NameNo.CaAxisNo.NGPush1].Io.DigitalInputs.1;

//负极踢废料
//arrAxisCtrl[NameNo.CaAxisNo.NGPush2].Io.DigitalInputs;
//arrAxisCtrl[NameNo.CaAxisNo.NGPush2].Io.biHomeSwitch:=NOT arrAxisCtrl[NameNo.CaAxisNo.NGPush2].Io.DigitalInputs.2;
//arrAxisCtrl[NameNo.CaAxisNo.NGPush2].Io.biNegLimit:=arrAxisCtrl[NameNo.CaAxisNo.NGPush2].Io.DigitalInputs.0;
//arrAxisCtrl[NameNo.CaAxisNo.NGPush2].Io.biPosLimit:=arrAxisCtrl[NameNo.CaAxisNo.NGPush2].Io.DigitalInputs.1;

//负极CCD压片升降
arrAxisCtrl[NameNo.CaAxisNo.CCDPressPush].Io.DigitalInputs;
arrAxisCtrl[NameNo.CaAxisNo.CCDPressPush].Io.biHomeSwitch:=NOT arrAxisCtrl[NameNo.CaAxisNo.CCDPressPush].Io.DigitalInputs.2;
//arrAxisCtrl[NameNo.CaAxisNo.CCDPressPush].Io.biNegLimit:=arrAxisCtrl[NameNo.CaAxisNo.CCDPressPush].Io.DigitalInputs.0;
//arrAxisCtrl[NameNo.CaAxisNo.CCDPressPush].Io.biPosLimit:=arrAxisCtrl[NameNo.CaAxisNo.CCDPressPush].Io.DigitalInputs.1;
END_ACTION

ACTION OutPut:
//输出映射	正极									
		Q101[1]	:=	arrCyCtrl[NameNo.AnCYNo.Inflation_L].Io.DOStatus1	;//	正极左放卷气涨轴张开				
		Q101[2]	:=	arrCyCtrl[NameNo.AnCYNo.Inflation_L].Io.DOStatus2	;//	正极左放卷气涨轴缩回				
		Q101[3]	:=	arrCyCtrl[NameNo.AnCYNo.Inflation_R].Io.DOStatus1	;//	正极右放卷气涨轴张开				
		Q101[4]	:=	arrCyCtrl[NameNo.AnCYNo.Inflation_R].Io.DOStatus2	;//	正极右放卷气涨轴缩回				
		Q101[5]	:=	arrCyCtrl[NameNo.AnCYNo.BoardPressL].Io.DOStatus1	;//	正极极片左接带气缸伸出				
		Q101[6]	:=	arrCyCtrl[NameNo.AnCYNo.BoardPressL].Io.DOStatus2	;//	正极极片左接带气缸缩回				
		Q101[7]	:=	arrCyCtrl[NameNo.AnCYNo.BoardPressR].Io.DOStatus1	;//	正极极片右接带气缸伸出				
		Q101[8]	:=	arrCyCtrl[NameNo.AnCYNo.BoardPressR].Io.DOStatus2	;//	正极极片右接带气缸缩回				
		Q101[9]	:=	arrCyCtrl[NameNo.AnEVNo.ConnectDustVacuo].Io.DOStatus1	;//	正极极片接带平台除尘真空打开				
		Q101[10]	:=	AnBtn.PoleBoxStartLight	;//	正极放卷启动按钮灯				
		Q101[11]	:=	AnBtn.CoderRollPressLight		;//	正极编码器压辊按钮灯			
		Q101[12]			;//					
		Q101[13]	:=	arrCyCtrl[NameNo.AnCYNo.DriverPressAux].Io.DOStatus1	;//	正极辅助驱动压辊伸出				
		Q101[14]	:=	arrCyCtrl[NameNo.AnCYNo.DriverPressAux].Io.DOStatus2	;//	正极辅助驱动压辊缩回				
		Q101[15]	:=	arrCyCtrl[NameNo.AnCYNo.CoderRollPress].Io.DOStatus1	;//	正极前线扫编码器压辊伸出				
		Q101[16]	:=	arrCyCtrl[NameNo.AnCYNo.CoderRollPress].Io.DOStatus2	;//	正极前线扫编码器压辊缩回				
										
		Q102[1]			;//					
		Q102[2]	:=	arrCyCtrl[NameNo.AnEVNo.LineSceneDustBlow].Io.DOStatus1	;//	正极线扫相机镜头除尘吹气				
		Q102[3]	:=	arrCyCtrl[NameNo.AnEVNo.LineSceneDustVacuo].Io.DOStatus1	;//	正极线扫相机镜头除尘真空				
		Q102[4]			;//					
		Q102[5]	:=	arrRecCtrl[NameNo.AnRecNo.PoleWind].Io.boManual	;//	正极放卷纠偏手动				
		Q102[6]	:=	arrRecCtrl[NameNo.AnRecNo.PoleWind].Io.boCentre	;//	正极放卷纠偏居中				
		Q102[7]	:=	arrRecCtrl[NameNo.AnRecNo.PoleWind].Io.boLock	;//	正极放卷纠偏外部锁定				
		Q102[8]	:=	arrRecCtrl[NameNo.AnRecNo.PoleWind].Io.boAuto	;//	正极放卷纠偏自动				
		Q102[9]	:=	arrRecCtrl[NameNo.AnRecNo.PoleProcess].Io.boManual	;//	正极行进纠偏手动				
		Q102[10]	:=	arrRecCtrl[NameNo.AnRecNo.PoleProcess].Io.boCentre	;//	正极行进纠偏居中				
		Q102[11]	:=	arrRecCtrl[NameNo.AnRecNo.PoleProcess].Io.boLock	;//	正极行进纠偏外部锁定				
		Q102[12]	:=	arrRecCtrl[NameNo.AnRecNo.PoleProcess].Io.boAuto	;//	正极行进纠偏自动				
		Q102[13]	:=	AnCCDIO.boChamferPhoto	;//	正极CCD冲R角定位拍照触发				
		Q102[14]	:=	AnCCDIO.boCuterPhoto	;//	正极CCD裁切定位拍照触发				
		Q102[15]	:=	AnCCDIO.boSizePhoto	;//	正极CCD尺寸检测拍照触发				
		Q102[16]			;//					
										
		Q103[1]	:=	arrCyCtrl[NameNo.AnCYNo.DriverPressDDR].Io.DOStatus1	;//	正极主驱动压辊伸出				
		Q103[2]	:=	arrCyCtrl[NameNo.AnCYNo.DriverPressDDR].Io.DOStatus2	;//	正极主驱动压辊缩回				
		Q103[3]	:=	AnBtn.DriverPressDDRLight	;//	正极主驱动压辊按钮灯				
		Q103[4]	:=	arrCyCtrl[NameNo.AnEVNo.AreaArrayDustBlow].Io.DOStatus1	;//	正极模切相机镜头除尘吹气				
		Q103[5]	:=	arrCyCtrl[NameNo.AnEVNo.MouldUpBlow].Io.DOStatus1	;//	正极模具上模吹气打开				
		Q103[6]	:=	arrCyCtrl[NameNo.AnEVNo.MouldDownVacuo].Io.DOStatus1	;//	正极模具下模真空				
		Q103[7]	:=	arrCyCtrl[NameNo.AnEVNo.MouldDownAir].Io.DOStatus1	;//	正极模具下模破真空				
		Q103[8]	:=	arrDustMotor[NameNo.AnMotorNo.CuterBeltDust].bo_Pul	;//	正极裁切输送皮带除尘毛刷正转				
		Q103[9]	:=	arrDustMotor[NameNo.AnMotorNo.CuterBeltDust].bo_Dir	;//	正极裁切输送皮带除尘毛刷反转				
		Q103[10]	:=	arrCyCtrl[NameNo.AnCYNo.NGRevBeltUpDown].Io.DOStatus1	;//	正极踢废倒装皮带升降气缸伸出				
		Q103[11]	:=	arrCyCtrl[NameNo.AnCYNo.NGRevBeltUpDown].Io.DOStatus2	;//	正极踢废倒装皮带升降气缸缩回				
		Q103[12]	:=	arrCyCtrl[NameNo.AnCYNo.NGRevBeltTension].Io.DOStatus1	;//	正极踢废倒装皮带1张紧气缸伸出				
		Q103[13]	:=	arrCyCtrl[NameNo.AnCYNo.NGRevBeltTension].Io.DOStatus2	;//	正极踢废倒装皮带1张紧气缸缩回				
		Q103[14]			;//					
		Q103[15]	:=	arrCyCtrl[NameNo.AnEVNo.ConnectDustVacuo].Io.DOStatus2	;//	正极极片接带平台除尘真空关闭					
		Q103[16]	:=	arrCyCtrl[NameNo.AnCYNo.WasteBoxPush].Io.DOStatus1	;//	正极连续废料收集箱推料气缸				
										
		Q104[1]	:=	arrDustMotor[NameNo.AnMotorNo.NGReverseBeltDust].bo_Pul	;//	正极踢废倒装皮带除尘毛刷正转				
		Q104[2]	:=	arrDustMotor[NameNo.AnMotorNo.NGReverseBeltDust].bo_Dir	;//	正极踢废倒装皮带除尘毛刷反转				
		//Q104[3]	:=	arrCyCtrl[NameNo.AnCYNo.NGBoxLock1].Io.DOStatus1	;//	正极NG收料1归正伸出				
		//Q104[4]	:=	arrCyCtrl[NameNo.AnCYNo.NGBoxLock1].Io.DOStatus2	;//	正极NG收料1归正缩回				
		//Q104[5]	:=	arrCyCtrl[NameNo.AnCYNo.NGBoxLock2].Io.DOStatus1	;//	正极NG收料2归正伸出				
		//Q104[6]	:=	arrCyCtrl[NameNo.AnCYNo.NGBoxLock2].Io.DOStatus2	;//	正极NG收料归正缩回				
		Q104[7]	:=	arrCyCtrl[NameNo.AnEVNo.NGPushInsideAir].Io.DOStatus1	;//	正极NG踢废腔室破真空				
		Q104[8]	:=	arrCyCtrl[NameNo.AnEVNo.NGPushInsideVacuo].Io.DOStatus1	;//	正极NG踢废腔室真空				
		Q104[9]	:=	AnsetpMotor.bo_Up	;//	正极NG料盒顶升上升				
		Q104[10]	:=	AnsetpMotor.bo_Down	;//	正极NG料盒顶升下降				
		Q104[11]	:=	AnBtn.NGBoxStartLight	;//	正极NG收料盒确认放入料框按钮灯				
		Q104[12]	:=	AnBtn.NGBoxMotor_JogUpLight	;//	正极NG收料盒电机上升按钮灯				
		Q104[13]	:=	AnBtn.NGBoxMotor_JogDownLight	;//	正极NG收料盒电机下降按钮灯				
		Q104[14]			;//					
		Q104[15]			;//					
		Q104[16]			;//					
										
		Q105[1]	:=	AnBtn.PoleBrushDustPush_ULight	;//	正极上表面毛刷除尘升降气缸按钮灯				
		Q105[2]	:=	AnBtn.PoleWindDustPush_ULight	;//	正极上表面超声波除尘升降气缸按钮灯				
		Q105[3]	:=	arrCyCtrl[NameNo.AnCYNo.PoleBrushDustPush_U].Io.DOStatus1	;//	正极上表面毛刷除尘升降气缸伸出				
		Q105[4]	:=	arrCyCtrl[NameNo.AnCYNo.PoleBrushDustPush_U].Io.DOStatus2	;//	正极上表面毛刷除尘升降气缸缩回				
		Q105[5]	:=	arrCyCtrl[NameNo.AnCYNo.PoleWindDustPush_U].Io.DOStatus1	;//	正极上表面风刀除尘升降气缸伸出				
		Q105[6]	:=	arrCyCtrl[NameNo.AnCYNo.PoleWindDustPush_U].Io.DOStatus2	;//	正极上表面风刀除尘升降气缸缩回				
		Q105[7]	:=	arrCyCtrl[NameNo.AnEVNo.BrushDustVacuo_U].Io.DOStatus1	;//	正极上表面毛刷除尘真空				
		Q105[8]	:=	arrCyCtrl[NameNo.AnEVNo.WindDustBlow_U].Io.DOStatus1	;//	正极上表面风刀除尘吹气				
		Q105[9]	:=	arrCyCtrl[NameNo.AnEVNo.WindDustVacuo_U].Io.DOStatus1	;//	正极上表面风刀除尘真空				
		Q105[10]	:=	arrDustMotor[NameNo.AnMotorNo.DedustBeltDust].bo_Pul	;//	正极上表面除尘皮带除尘毛刷正转				
		Q105[11]	:=	arrDustMotor[NameNo.AnMotorNo.DedustBeltDust].bo_Dir	;//	正极上表面除尘皮带除尘毛刷反转				
		Q105[12]	:=	arrDustMotor[NameNo.AnMotorNo.PoleBrushDust_U].bo_Pul	;//	正极上表面极片除尘毛刷正转				
		Q105[13]	:=	arrDustMotor[NameNo.AnMotorNo.PoleBrushDust_U].bo_Dir	;//	正极上表面极片除尘毛刷反转				
		Q105[14]	:=	arrDustMotor[NameNo.AnMotorNo.DDR_Dust].bo_Pul		;//	正极主驱辊除尘毛刷正转				
		Q105[15]	:=	arrDustMotor[NameNo.AnMotorNo.DDR_Dust].bo_Dir		;//	正极主驱辊除尘毛刷反转				
		Q105[16]			;//					
										
		Q106[1]	:=	AnBtn.PoleBrushDustPush_DLight	;//	正极下表面毛刷除尘升降气缸按钮灯				
		Q106[2]	:=	AnBtn.PoleWindDustPush_DLight	;//	正极下表面超声波除尘升降气缸按钮灯				
		Q106[3]	:=	arrCyCtrl[NameNo.AnCYNo.PoleBrushDustPush_D].Io.DOStatus1	;//	正极下表面毛刷除尘升降气缸伸出				
		Q106[4]	:=	arrCyCtrl[NameNo.AnCYNo.PoleBrushDustPush_D].Io.DOStatus2	;//	正极下表面毛刷除尘升降气缸缩回				
		Q106[5]	:=	arrCyCtrl[NameNo.AnCYNo.PoleWindDustPush_D].Io.DOStatus1	;//	正极下表面风刀除尘升降气缸伸出				
		Q106[6]	:=	arrCyCtrl[NameNo.AnCYNo.PoleWindDustPush_D].Io.DOStatus2	;//	正极下表面风刀除尘升降气缸缩回				
		Q106[7]	:=	arrCyCtrl[NameNo.AnCYNo.DustRevBeltUpDown].Io.DOStatus1	;//	正极下表面除尘倒装皮带升降气缸伸出				
		Q106[8]	:=	arrCyCtrl[NameNo.AnCYNo.DustRevBeltUpDown].Io.DOStatus2	;//	正极下表面除尘倒装皮带升降气缸缩回				
		Q106[9]	:=	arrCyCtrl[NameNo.AnEVNo.BrushDustVacuo_D].Io.DOStatus1	;//	正极下表面毛刷除尘真空				
		Q106[10]	:=	arrCyCtrl[NameNo.AnEVNo.WindDustBlow_D].Io.DOStatus1	;//	正极下表面风刀除尘吹气				
		Q106[11]	:=	arrCyCtrl[NameNo.AnEVNo.WindDustVacuo_D].Io.DOStatus1	;//	正极下表面风刀除尘真空				
		Q106[12]	:=	arrDustMotor[NameNo.AnMotorNo.DedustReverseBeltDust].bo_Pul	;//	正极下表面除尘皮带除尘毛刷正转				
		Q106[13]	:=	arrDustMotor[NameNo.AnMotorNo.DedustReverseBeltDust].bo_Dir	;//	正极下表面除尘皮带除尘毛刷反转				
		Q106[14]	:=	arrDustMotor[NameNo.AnMotorNo.PoleBrushDust_D].bo_Pul	;//	正极下表面极片除尘毛刷正转				
		Q106[15]	:=	arrDustMotor[NameNo.AnMotorNo.PoleBrushDust_D].bo_Dir	;//	正极下表面极片除尘毛刷反转				
		Q106[16]			;//					
										
		Q107[1]	:=	AnSys.boStartLight	;//	正极控制面板启动按钮灯				
		Q107[2]	:=	AnSys.boResetLight	;//	正极控制面板复位按钮灯				
		Q107[3]	:=	AnSys.boStopLight	;//	正极控制面板停止按钮灯				
		Q107[4]	:=	stSysState.boYellowLight	;//	正极三色灯_黄				
		Q107[5]	:=	stSysState.boGreenLight	;//	正极三色灯_绿				
		Q107[6]	:=	stSysState.boRedLight	;//	正极三色灯_红				
		Q107[7]	:=	stSysState.boBuzzer AND NOT ProductPar.iModeEN.bBuzzerEN	;//	正极三色灯_蜂鸣器				
		Q107[8]			;//					
		Q107[9]	:=	arrCyCtrl[NameNo.AnEVNo.RJ_Blow].Io.DOStatus1		;//	正极R角吹气		
		Q107[10]	:=	arrCyCtrl[NameNo.AnEVNo.RJDustBlow].Io.DOStatus1		;//R角风刀吹气			
		Q107[11]			;//	正极激光指示器				
		Q107[12]			;//					
		Q107[13]			;//					
		Q107[14]			;//					
		Q107[15]			;//					
		Q107[16]			;//					
										
		Q108[1]			;//					
		Q108[2]	:=AnCCDIO.boXSPhoto OR  AnCCDIO.hmiXSPhoto		;//			
		Q108[3]			;//					
		Q108[4]			;//					
		Q108[5]			;//					
		Q108[6]			;//					
		Q108[7]			;//					
		Q108[8]			;//					
		Q108[9]			;//					
		Q108[10]			;//					
		Q108[11]			;//					
		Q108[12]			;//					
		Q108[13]			;//					
		Q108[14]			;//					
		Q108[15]			;//					
		Q108[16]			;//					
										
		Q109[1]	:=	bytePower.0	;//	正极模切电源				
		Q109[2]	:=	bytePower.1	;//	负极模切电源				
		Q109[3]	:=	bytePower.2	;//	叠台1电源				
		Q109[4]	:=	bytePower.3	;//	叠台2电源				
		Q109[5]	:=	bytePower.4	;//	叠台3电源				
		Q109[6]	:=	bytePower.5	;//	后段滤波器电源				
		Q109[7]	:=	bytePower.6	;//	后段加热回路电源				
		Q109[8]			;//					
		Q109[9]			;//					
		Q109[10]			;//					
		Q109[11]			;//					
		Q109[12]			;//					
		Q109[13]			;//					
		Q109[14]			;//					
		Q109[15]			;//					
		Q109[16]			;//					
										
//输出映射	负极									
		Q201[1]	:=	arrCyCtrl[NameNo.CaCYNo.Inflation_L].Io.DOStatus1	;//	负极左放卷气涨轴张开				
		Q201[2]	:=	arrCyCtrl[NameNo.CaCYNo.Inflation_L].Io.DOStatus2	;//	负极左放卷气涨轴缩回				
		Q201[3]	:=	arrCyCtrl[NameNo.CaCYNo.Inflation_R].Io.DOStatus1	;//	负极右放卷气涨轴张开				
		Q201[4]	:=	arrCyCtrl[NameNo.CaCYNo.Inflation_R].Io.DOStatus2	;//	负极右放卷气涨轴缩回				
		Q201[5]	:=	arrCyCtrl[NameNo.CaCYNo.BoardPressL].Io.DOStatus1	;//	负极极片左接带气缸伸出				
		Q201[6]	:=	arrCyCtrl[NameNo.CaCYNo.BoardPressL].Io.DOStatus2	;//	负极极片左接带气缸缩回				
		Q201[7]	:=	arrCyCtrl[NameNo.CaCYNo.BoardPressR].Io.DOStatus1	;//	负极极片右接带气缸伸出				
		Q201[8]	:=	arrCyCtrl[NameNo.CaCYNo.BoardPressR].Io.DOStatus2	;//	负极极片右接带气缸缩回				
		Q201[9]	:=	arrCyCtrl[NameNo.CaEVNo.ConnectDustVacuo].Io.DOStatus1	;//	负极极片接带平台除尘真空打开				
		Q201[10]	:=	CaBtn.PoleBoxStartLight	;//	负极放卷启动按钮灯				
		Q201[11]	:=	CaBtn.CoderRollPressLight		;//	负极编码器压辊按钮灯		;//	
		Q201[12]			;//					
		Q201[13]	:=	arrCyCtrl[NameNo.CaCYNo.DriverPressAux].Io.DOStatus1	;//	负极辅助驱动压辊伸出				
		Q201[14]	:=	arrCyCtrl[NameNo.CaCYNo.DriverPressAux].Io.DOStatus2	;//	负极辅助驱动压辊缩回				
		Q201[15]	:=	arrCyCtrl[NameNo.CaCYNo.CoderRollPress].Io.DOStatus1	;//	负极前线扫编码器压辊伸出				
		Q201[16]	:=	arrCyCtrl[NameNo.CaCYNo.CoderRollPress].Io.DOStatus2	;//	负极前线扫编码器压辊缩回				
										
		Q202[1]			;//					
		Q202[2]	:=	arrCyCtrl[NameNo.CaEVNo.LineSceneDustBlow].Io.DOStatus1	;//	负极线扫相机镜头除尘吹气				
		Q202[3]	:=	arrCyCtrl[NameNo.CaEVNo.LineSceneDustVacuo].Io.DOStatus1	;//	负极线扫相机镜头除尘真空				
		Q202[4]			;//					
		Q202[5]	:=	arrRecCtrl[NameNo.CaRecNo.PoleWind].Io.boManual	;//	负极放卷纠偏手动				
		Q202[6]	:=	arrRecCtrl[NameNo.CaRecNo.PoleWind].Io.boCentre	;//	负极放卷纠偏居中				
		Q202[7]	:=	arrRecCtrl[NameNo.CaRecNo.PoleWind].Io.boLock	;//	负极放卷纠偏外部锁定				
		Q202[8]	:=	arrRecCtrl[NameNo.CaRecNo.PoleWind].Io.boAuto	;//	负极放卷纠偏自动				
		Q202[9]	:=	arrRecCtrl[NameNo.CaRecNo.PoleProcess].Io.boManual	;//	负极行进纠偏手动				
		Q202[10]	:=	arrRecCtrl[NameNo.CaRecNo.PoleProcess].Io.boCentre	;//	负极行进纠偏居中				
		Q202[11]	:=	arrRecCtrl[NameNo.CaRecNo.PoleProcess].Io.boLock	;//	负极行进纠偏外部锁定				
		Q202[12]	:=	arrRecCtrl[NameNo.CaRecNo.PoleProcess].Io.boAuto	;//	负极行进纠偏自动				
		Q202[13]	:=	CaCCDIO.boChamferPhoto	;//	负极CCD冲R角定位拍照触发				
		Q202[14]	:=	CaCCDIO.boCuterPhoto	;//	负极CCD裁切定位拍照触发				
		Q202[15]	:=	CaCCDIO.boSizePhoto	;//	负极CCD尺寸检测拍照触发				
		Q202[16]			;//					
										
		Q203[1]	:=	arrCyCtrl[NameNo.CaCYNo.DriverPressDDR].Io.DOStatus1	;//	负极主驱动压辊伸出				
		Q203[2]	:=	arrCyCtrl[NameNo.CaCYNo.DriverPressDDR].Io.DOStatus2	;//	负极主驱动压辊缩回				
		Q203[3]	:=	CaBtn.DriverPressDDRLight	;//	负极主驱动压辊按钮灯				
		Q203[4]	:=	arrCyCtrl[NameNo.CaEVNo.AreaArrayDustBlow].Io.DOStatus1	;//	负极模切相机镜头除尘吹气				
		Q203[5]	:=	arrCyCtrl[NameNo.CaEVNo.MouldUpBlow].Io.DOStatus1	;//	负极模具上模吹气打开				
		Q203[6]	:=	arrCyCtrl[NameNo.CaEVNo.MouldDownVacuo].Io.DOStatus1	;//	负极模具下模真空				
		Q203[7]	:=	arrCyCtrl[NameNo.CaEVNo.MouldDownAir].Io.DOStatus1	;//	负极模具下模破真空				
		Q203[8]	:=	arrDustMotor[NameNo.CaMotorNo.CuterBeltDust].bo_Pul	;//	负极裁切输送皮带除尘毛刷正转				
		Q203[9]	:=	arrDustMotor[NameNo.CaMotorNo.CuterBeltDust].bo_Dir	;//	负极裁切输送皮带除尘毛刷反转				
		Q203[10]	:=	arrCyCtrl[NameNo.CaCYNo.NGRevBeltUpDown].Io.DOStatus1	;//	负极踢废倒装皮带升降气缸伸出				
		Q203[11]	:=	arrCyCtrl[NameNo.CaCYNo.NGRevBeltUpDown].Io.DOStatus2	;//	负极踢废倒装皮带升降气缸缩回				
		Q203[12]	:=	arrCyCtrl[NameNo.CaCYNo.NGRevBeltTension].Io.DOStatus1	;//	负极踢废倒装皮带1张紧气缸伸出				
		Q203[13]	:=	arrCyCtrl[NameNo.CaCYNo.NGRevBeltTension].Io.DOStatus2	;//	负极踢废倒装皮带1张紧气缸缩回				
		Q203[14]			;//					
		Q203[15]	:=	arrCyCtrl[NameNo.CaEVNo.ConnectDustVacuo].Io.DOStatus2	;//	负极极片接带平台除尘真空关闭			;//					
		Q203[16]	:=	arrCyCtrl[NameNo.CaCYNo.WasteBoxPush].Io.DOStatus1	;//	负极连续废料收集箱推料气缸				
										
		Q204[1]	:=	arrDustMotor[NameNo.CaMotorNo.NGReverseBeltDust].bo_Pul	;//	负极踢废倒装皮带除尘毛刷正转				
		Q204[2]	:=	arrDustMotor[NameNo.CaMotorNo.NGReverseBeltDust].bo_Dir	;//	负极踢废倒装皮带除尘毛刷反转				
		//Q204[3]	:=	arrCyCtrl[NameNo.CaCYNo.NGBoxLock1].Io.DOStatus1	;//	负极NG收料1归正伸出				
		//Q204[4]	:=	arrCyCtrl[NameNo.CaCYNo.NGBoxLock1].Io.DOStatus2	;//	负极NG收料1归正缩回				
		//Q204[5]	:=	arrCyCtrl[NameNo.CaCYNo.NGBoxLock2].Io.DOStatus1	;//	负极NG收料2归正伸出				
		//Q204[6]	:=	arrCyCtrl[NameNo.CaCYNo.NGBoxLock2].Io.DOStatus2	;//	负极NG收料归正缩回				
		Q204[7]	:=	arrCyCtrl[NameNo.CaEVNo.NGPushInsideAir].Io.DOStatus1	;//	负极NG踢废腔室破真空				
		Q204[8]	:=	arrCyCtrl[NameNo.CaEVNo.NGPushInsideVacuo].Io.DOStatus1	;//	负极NG踢废腔室真空				
		Q204[9]	:=	CasetpMotor.bo_Up	;//	负极NG料盒顶升上升				
		Q204[10]	:=	CasetpMotor.bo_Down	;//	负极NG料盒顶升下降				
		Q204[11]	:=	CaBtn.NGBoxStartLight	;//	负极NG收料盒确认放入料框按钮灯				
		Q204[12]	:=	CaBtn.NGBoxMotor_JogUpLight	;//	负极NG收料盒电机上升按钮灯				
		Q204[13]	:=	CaBtn.NGBoxMotor_JogDownLight	;//	负极NG收料盒电机下降按钮灯				
		Q204[14]			;//					
		Q204[15]			;//					
		Q204[16]			;//					
										
		Q205[1]	:=	CaBtn.PoleBrushDustPush_ULight	;//	负极上表面毛刷除尘升降气缸按钮灯				
		Q205[2]	:=	CaBtn.PoleWindDustPush_ULight	;//	负极上表面超声波除尘升降气缸按钮灯				
		Q205[3]	:=	arrCyCtrl[NameNo.CaCYNo.PoleBrushDustPush_U].Io.DOStatus1	;//	负极上表面毛刷除尘升降气缸伸出				
		Q205[4]	:=	arrCyCtrl[NameNo.CaCYNo.PoleBrushDustPush_U].Io.DOStatus2	;//	负极上表面毛刷除尘升降气缸缩回				
		Q205[5]	:=	arrCyCtrl[NameNo.CaCYNo.PoleWindDustPush_U].Io.DOStatus1	;//	负极上表面风刀除尘升降气缸伸出				
		Q205[6]	:=	arrCyCtrl[NameNo.CaCYNo.PoleWindDustPush_U].Io.DOStatus2	;//	负极上表面风刀除尘升降气缸缩回				
		Q205[7]	:=	arrCyCtrl[NameNo.CaEVNo.BrushDustVacuo_U].Io.DOStatus1	;//	负极上表面毛刷除尘真空				
		Q205[8]	:=	arrCyCtrl[NameNo.CaEVNo.WindDustBlow_U].Io.DOStatus1	;//	负极上表面风刀除尘吹气				
		Q205[9]	:=	arrCyCtrl[NameNo.CaEVNo.WindDustVacuo_U].Io.DOStatus1	;//	负极上表面风刀除尘真空				
		Q205[10]	:=	arrDustMotor[NameNo.CaMotorNo.DedustBeltDust].bo_Pul	;//	负极上表面除尘皮带除尘毛刷正转				
		Q205[11]	:=	arrDustMotor[NameNo.CaMotorNo.DedustBeltDust].bo_Dir	;//	负极上表面除尘皮带除尘毛刷反转				
		Q205[12]	:=	arrDustMotor[NameNo.CaMotorNo.PoleBrushDust_U].bo_Pul	;//	负极上表面极片除尘毛刷正转				
		Q205[13]	:=	arrDustMotor[NameNo.CaMotorNo.PoleBrushDust_U].bo_Dir	;//	负极上表面极片除尘毛刷反转				
		Q205[14]	:=	arrDustMotor[NameNo.CaMotorNo.DDR_Dust].bo_Pul	;//	负极主驱辊除尘毛刷正转					
		Q205[15]	:=	arrDustMotor[NameNo.CaMotorNo.DDR_Dust].bo_Dir	;//	负极主驱辊除尘毛刷正转			;//					
		Q205[16]			;//					
										
		Q206[1]	:=	CaBtn.PoleBrushDustPush_DLight	;//	负极下表面毛刷除尘升降气缸按钮灯				
		Q206[2]	:=	CaBtn.PoleWindDustPush_DLight	;//	负极下表面超声波除尘升降气缸按钮灯				
		Q206[3]	:=	arrCyCtrl[NameNo.CaCYNo.PoleBrushDustPush_D].Io.DOStatus1	;//	负极下表面毛刷除尘升降气缸伸出				
		Q206[4]	:=	arrCyCtrl[NameNo.CaCYNo.PoleBrushDustPush_D].Io.DOStatus2	;//	负极下表面毛刷除尘升降气缸缩回				
		Q206[5]	:=	arrCyCtrl[NameNo.CaCYNo.PoleWindDustPush_D].Io.DOStatus1	;//	负极下表面风刀除尘升降气缸伸出				
		Q206[6]	:=	arrCyCtrl[NameNo.CaCYNo.PoleWindDustPush_D].Io.DOStatus2	;//	负极下表面风刀除尘升降气缸缩回				
		Q206[7]	:=	arrCyCtrl[NameNo.CaCYNo.DustRevBeltUpDown].Io.DOStatus1	;//	负极下表面除尘倒装皮带升降气缸伸出				
		Q206[8]	:=	arrCyCtrl[NameNo.CaCYNo.DustRevBeltUpDown].Io.DOStatus2	;//	负极下表面除尘倒装皮带升降气缸缩回				
		Q206[9]	:=	arrCyCtrl[NameNo.CaEVNo.BrushDustVacuo_D].Io.DOStatus1	;//	负极下表面毛刷除尘真空				
		Q206[10]	:=	arrCyCtrl[NameNo.CaEVNo.WindDustBlow_D].Io.DOStatus1	;//	负极下表面风刀除尘吹气				
		Q206[11]	:=	arrCyCtrl[NameNo.CaEVNo.WindDustVacuo_D].Io.DOStatus1	;//	负极下表面风刀除尘真空				
		Q206[12]	:=	arrDustMotor[NameNo.CaMotorNo.DedustReverseBeltDust].bo_Pul	;//	负极下表面除尘皮带除尘毛刷正转				
		Q206[13]	:=	arrDustMotor[NameNo.CaMotorNo.DedustReverseBeltDust].bo_Dir	;//	负极下表面除尘皮带除尘毛刷反转				
		Q206[14]	:=	arrDustMotor[NameNo.CaMotorNo.PoleBrushDust_D].bo_Pul	;//	负极下表面极片除尘毛刷正转				
		Q206[15]	:=	arrDustMotor[NameNo.CaMotorNo.PoleBrushDust_D].bo_Dir	;//	负极下表面极片除尘毛刷反转				
		Q206[16]			;//					
										
		Q207[1]	:=	CaSys.boStartLight	;//	负极控制面板启动按钮灯				
		Q207[2]	:=	CaSys.boResetLight	;//	负极控制面板复位按钮灯				
		Q207[3]	:=	CaSys.boStopLight	;//	负极控制面板停止按钮灯				
		Q207[4]	:=	stSysState.boYellowLight	;//	负极三色灯_黄				
		Q207[5]	:=	stSysState.boGreenLight	;//	负极三色灯_绿				
		Q207[6]	:=	stSysState.boRedLight	;//	负极三色灯_红				
		Q207[7]	:=	stSysState.boBuzzer AND NOT ProductPar.iModeEN.bBuzzerEN	;//	负极三色灯_蜂鸣器				
		Q207[8]				;//		
		Q207[9]	:=	arrCyCtrl[NameNo.CaEVNo.RJ_Blow].Io.DOStatus1		;//	负极R角吹气					
		Q207[10]	:=	arrCyCtrl[NameNo.CaEVNo.RJDustBlow].Io.DOStatus1		;//R角风刀吹气		
		Q207[11]			;//	负极激光指示器				
		Q207[12]			;//					
		Q207[13]			;//					
		Q207[14]			;//					
		Q207[15]			;//					
		Q207[16]			;//					
										
		Q208[1]			;//					
		Q208[2]:=CaCCDIO.boXSPhoto OR	 CaCCDIO.hmiXSPhoto	;//			
		Q208[3]			;//					
		Q208[4]			;//					
		Q208[5]			;//					
		Q208[6]			;//					
		Q208[7]			;//					
		Q208[8]			;//					
		Q208[9]			;//					
		Q208[10]			;//					
		Q208[11]			;//					
		Q208[12]			;//					
		Q208[13]			;//					
		Q208[14]			;//					
		Q208[15]			;//					
		Q208[16]			;//					
										
		Q209[1]			;//					
		Q209[2]			;//					
		Q209[3]			;//					
		Q209[4]			;//					
		Q209[5]			;//					
		Q209[6]			;//					
		Q209[7]			;//					
		Q209[8]			;//					
		Q209[9]			;//					
		Q209[10]			;//					
		Q209[11]			;//					
		Q209[12]			;//					
		Q209[13]			;//					
		Q209[14]			;//					
		Q209[15]			;//					
		Q209[16]			;//		


Q30103	:=	arrDustMotor[NameNo.AnMotorNo.FeduanbeltDust1].bo_Pul ;//正极模切分段皮带1除尘毛刷正转
Q30104	:=	arrDustMotor[NameNo.AnMotorNo.FeduanbeltDust1].bo_Dir ;//正极模切分段皮带1除尘毛刷反转
Q30201	:=	arrDustMotor[NameNo.CaMotorNo.FeduanbeltDust1].bo_Pul ;//正极模切分段皮带1除尘毛刷正转
Q30202  :=	arrDustMotor[NameNo.CaMotorNo.FeduanbeltDust1].bo_Dir;//正极模切分段皮带1除尘毛刷反转

Q40103	:=	arrDustMotor[NameNo.AnMotorNo.FeduanbeltDust2].bo_Pul ;//正极模切分段皮带2除尘毛刷正转
Q40104	:=	arrDustMotor[NameNo.AnMotorNo.FeduanbeltDust2].bo_Dir ;//正极模切分段皮带2除尘毛刷反转
Q40201	:=	arrDustMotor[NameNo.CaMotorNo.FeduanbeltDust2].bo_Pul ;//正极模切分段皮带2除尘毛刷正转
Q40202	:=	arrDustMotor[NameNo.CaMotorNo.FeduanbeltDust2].bo_Dir ;//正极模切分段皮带2除尘毛刷反转

Q50103	:=	arrDustMotor[NameNo.AnMotorNo.FeduanbeltDust3].bo_Pul ;//正极模切分段皮带3除尘毛刷正转
Q50104	:=	arrDustMotor[NameNo.AnMotorNo.FeduanbeltDust3].bo_Dir ;//正极模切分段皮带3除尘毛刷反转
Q50201	:=	arrDustMotor[NameNo.CaMotorNo.FeduanbeltDust3].bo_Pul ;//正极模切分段皮带3除尘毛刷正转
Q50202	:=	arrDustMotor[NameNo.CaMotorNo.FeduanbeltDust3].bo_Dir ;//正极模切分段皮带3除尘毛刷反转
END_ACTION

END_PROGRAM

// ---- POUs/BasicFunction/Basic/01_IO/FB_Filter_ADV2.TcPOU
FUNCTION_BLOCK FB_Filter_ADV2   //模拟量输入转换
VAR_INPUT
	iMode        :INT;//数据转换模式  1：周期平均   2：实时平均    3：无处理
    AD           :INT;
	iLimitH      :REAL;//转换前高限值
	iLimitL      :REAL;//转换前低限值
	fRangeH      :REAL;//量程高限
	fRangeL      :REAL;//量程低限
	fPointNum    :INT;//采集次数

	
END_VAR
VAR_OUTPUT
	Out_Value    :REAL;//转换输出

END_VAR
VAR
	i	            :INT;	
	Dgt_in	        :REAL;	
	Mid_Volt	    :REAL;	
	New_Period	    :INT;	
	iSetp	        :INT:=88;	
	fSumAdIn	    :REAL;	
	Ad_inputArray	:ARRAY[0..4000] OF REAL	;	//均值滤波数组
	K1	            :INT;	
	faverageValue	:REAL;	
	I2: INT;
END_VAR



IF iSetp=88 THEN
	IF iLimitH>0 AND fRangeH<>0 AND fPointNum>2 AND fPointNum<=4000 THEN
		fSumAdIn:=0;
		IF iMode=1 THEN         //1：周期平均
			// Clear(InOut:=Ad_inputArray);
			 MEMSET(ADR(Ad_inputArray),0,SIZEOF(Ad_inputArray));
			 i:=1;
			iSetp:=10;
		ELSIF iMode=2 THEN    // 2：实时平均  
			I2:=1;
			iSetp:=20;	
		ELSIF iMode=3 THEN    //3：无处理
			  iSetp:=30;	
		END_IF;
	END_IF;
END_IF

IF iSetp=10 THEN
   Ad_inputArray[i]:=INT_TO_REAL(AD);
	i:=i+1;
	IF i>fPointNum THEN
		 iSetp:=11;	
	END_IF;	
END_IF

IF iSetp=11 THEN
	FOR K1:=1 TO fPointNum BY 1 DO 
		  fSumAdIn:=fSumAdIn+Ad_inputArray[K1];
	END_FOR;
	faverageValue:=fSumAdIn/fPointNum; //平均AD转换值
	IF iLimitH-iLimitL<>0 THEN
		Out_Value:=( (faverageValue- iLimitL) * (fRangeH-fRangeL))/ (iLimitH-iLimitL)+fRangeL;
	END_IF
	iSetp:=88;
END_IF



CASE   iSetp OF 
 // 2：实时平均  	
20:
	Ad_inputArray[0]:=INT_TO_REAL(AD);
	FOR K1:=1 TO fPointNum BY 1 DO 
				IF K1<=fPointNum THEN 
					Ad_inputArray[fPointNum+1-K1]:=Ad_inputArray[fPointNum-K1];
			  END_IF; 
	END_FOR;
	iSetp:=21;
21:
    I2:=I2+1;
    IF I2>fPointNum THEN
        	iSetp:=22;
	ELSE
	  	iSetp:=20;
	END_IF
22:
	FOR K1:=1 TO fPointNum BY 1 DO 
		  fSumAdIn:=fSumAdIn+Ad_inputArray[K1];
	END_FOR;
	faverageValue:=fSumAdIn/fPointNum; //平均AD转换值
	//Out_Value:=( (faverageValue-INT_TO_REAL( iLimitL)) * (fRangeH-fRangeL))/ (INT_TO_REAL( iLimitH)-INT_TO_REAL( iLimitL))+fRangeL;
	IF iLimitH-iLimitL<>0 THEN
		Out_Value:=( (faverageValue- iLimitL) * (fRangeH-fRangeL))/ (iLimitH-iLimitL)+fRangeL;
	END_IF 
	iSetp:=88;
	
END_CASE




IF iSetp=30 THEN
	faverageValue:=INT_TO_REAL(AD);
	//Out_Value:=( (faverageValue-INT_TO_REAL( iLimitL)) * (fRangeH-fRangeL))/ (INT_TO_REAL( iLimitH)-INT_TO_REAL( iLimitL))+fRangeL;
	IF iLimitH-iLimitL<>0 THEN
     	Out_Value:=( (faverageValue- iLimitL) * (fRangeH-fRangeL))/ (iLimitH-iLimitL)+fRangeL;
	END_IF
	iSetp:=88;
END_IF






(*

IF iSetp=88 THEN
	IF iLimitH>0 AND fRangeH<>0 AND fPointNum>2 AND fPointNum<=20 THEN
		fSumAdIn:=0;
		IF iMode=1 THEN         //1：周期平均
			// Clear(InOut:=Ad_inputArray);
			 MEMSET(ADR(Ad_inputArray),0,SIZEOF(Ad_inputArray));
			 i:=1;
			iSetp:=10;
		ELSIF iMode=2 THEN    // 2：实时平均  
			iSetp:=20;	
		ELSIF iMode=3 THEN    //3：无处理
			  iSetp:=30;	
		END_IF;
	END_IF;
END_IF

IF iSetp=10 THEN
   Ad_inputArray[i]:=INT_TO_REAL(AD);
	i:=i+1;
	IF i>fPointNum THEN
		 iSetp:=11;	
	END_IF;	
END_IF

IF iSetp=11 THEN
	FOR K1:=1 TO fPointNum BY 1 DO 
		  fSumAdIn:=fSumAdIn+Ad_inputArray[K1];
	END_FOR;
	faverageValue:=fSumAdIn/fPointNum; //平均AD转换值
	IF iLimitH-iLimitL<>0 THEN
		Out_Value:=( (faverageValue- iLimitL) * (fRangeH-fRangeL))/ (iLimitH-iLimitL)+fRangeL;
	END_IF
	iSetp:=88;
END_IF

IF iSetp=20 THEN
	Ad_inputArray[0]:=INT_TO_REAL(AD);
	FOR K1:=1 TO fPointNum BY 1 DO 
				IF K1<=fPointNum THEN 
					Ad_inputArray[fPointNum+1-K1]:=Ad_inputArray[fPointNum-K1];
			  END_IF; 
	END_FOR;
	iSetp:=21;
END_IF

IF iSetp=21 THEN
	FOR K1:=1 TO fPointNum BY 1 DO 
		  fSumAdIn:=fSumAdIn+Ad_inputArray[K1];
	END_FOR;
	faverageValue:=fSumAdIn/fPointNum; //平均AD转换值
	//Out_Value:=( (faverageValue-INT_TO_REAL( iLimitL)) * (fRangeH-fRangeL))/ (INT_TO_REAL( iLimitH)-INT_TO_REAL( iLimitL))+fRangeL;
	IF iLimitH-iLimitL<>0 THEN
		Out_Value:=( (faverageValue- iLimitL) * (fRangeH-fRangeL))/ (iLimitH-iLimitL)+fRangeL;
	END_IF 
	iSetp:=88;
END_IF

IF iSetp=30 THEN
	faverageValue:=INT_TO_REAL(AD);
	//Out_Value:=( (faverageValue-INT_TO_REAL( iLimitL)) * (fRangeH-fRangeL))/ (INT_TO_REAL( iLimitH)-INT_TO_REAL( iLimitL))+fRangeL;
	IF iLimitH-iLimitL<>0 THEN
     	Out_Value:=( (faverageValue- iLimitL) * (fRangeH-fRangeL))/ (iLimitH-iLimitL)+fRangeL;
	END_IF
	iSetp:=88;
END_IF

*)

END_FUNCTION_BLOCK

// ---- POUs/BasicFunction/Data/FC_Filter_AA.TcPOU
FUNCTION FC_Filter_AA : REAL
VAR_INPUT
	SclIn:REAL;
	X0:REAL;
	Y0:REAL;
	X1:REAL;
	Y1:REAL;
END_VAR
VAR
END_VAR

IF X1-X0>0 AND Y1-Y0>0 THEN
	IF SclIn>=X0 AND SclIn<=X1 THEN
		FC_Filter_AA:=((Y1-Y0)*(SclIn-X0))/(X1-X0)+Y0;
	ELSIF SclIn<X0 THEN	
		FC_Filter_AA:=Y0;
	ELSIF SclIn>X1 THEN
		FC_Filter_AA:=Y1;
	END_IF 
END_IF

END_FUNCTION

// ---- POUs/POUs/MainState.TcPOU
PROGRAM MainState
VAR
	iMainSetp :INT;
	I1: UINT;
	iErrorSetp: INT;
	iLightSel: INT;
	bTurnOn: BOOL;
	bDoor_Stop: BOOL;
	I2: INT;
	I4: INT;
	I5: INT;
	i: UINT;
	iCode2: ICode;
	ExtSetVel: LREAL;
	ExtSetPos: LREAL;
	ExtSetAcc: LREAL;
	ExtSetDec: DINT;
	InitSetp: INT;
	rtStoping: R_TRIG;
	iMainInitSetp: INT;
	iMainEStopSetp: INT;
	K1: UINT;
	bInitReset: BOOL;
	DA1: INT;
	Code1: BOOL;
	Code2: BOOL;
	Code3: BOOL;
	Code4: BOOL;
	CyCtrl: INT;
	bWaterOn: BOOL;
	
	Execute: BOOL;
	bCoeWrite_GlueFeed: BOOL;
	bWaterOn2: BOOL;
	arrError:					ARRAY[1..10]OF BOOL;
	bEncloserEstop:BOOL;//外罩急停汇总
	bBoxEstop:BOOL;//按钮盒急停汇总
	F: INT;
	D195: MS_Alarm;
	D196: MS_Alarm;
	D197: MS_Alarm;
	D198: MS_Alarm;
	D199: MS_Alarm;
	D200: MS_Alarm;
	D201: MS_Alarm;
	D202: MS_Alarm;
	D203: MS_Alarm;
	D204: MS_Alarm;
	D205: MS_Alarm;
	D206: MS_Alarm;
	AnFD1: MS_Alarm;
	AnFD2: MS_Alarm;
	AnFD3: MS_Alarm;
	CaFD1: MS_Alarm;
	CaFD2: MS_Alarm;
	CaFD3: MS_Alarm;
	K2:INT;
	tCycleTimer: TON;
	bSave: BOOL;
	testii2: INT;
	bReadDataFirstCyle: BOOL;
	bReadDataCyle2: BOOL;
	bSaveTest: BOOL;
	rtSaveData: R_TRIG;
	CleanTrig: R_TRIG;
	CaCibang: R_TRIG;
	AnCibang: R_TRIG;
	CaCleanBrush:R_TRIG;
	AnCleanBrush:R_TRIG;
	
END_VAR

VAR
	R_TRIG_Bt: 			ARRAY[1..10]OF R_TRIG;
	TON20:Tc2_Standard.TON;	
//	TON21:Tc2_Standard.TON;	
	rt100:Tc2_Standard.R_TRIG;
	rt101:Tc2_Standard.R_TRIG;

	tDelayBuzze:TON;
	FanTon:TON;//除尘风机计时
	FanTonS:REAL;//除尘风机寿命秒
	FanTonH:REAL;//除尘风机寿命小时
	FanTonH_Set:REAL;//除尘风机寿命设定小时
	aAirAlarm_TON:TON;//气压报警延时；
	aTime:ARRAY[1..99] OF TON;//延时备用，1-16风速仪报警延时；
	aAlarm:ARRAY[1..99] OF BOOL;//报警预留;   1、气压不足报警；2、正极R角清废料报警；3、负极R角清废料报警；4、正极R角清废料计数错误；5、负极R角清废料计数错误；6、风机未启用报警；7、风机故障报警； 16-19、安全光栅报警；20-29、风速仪报警；30-47毛刷旋转感应报警，48毛刷旋转感应报警汇总,50:模切通道安全门报警；
	RT200:ARRAY[1..4] OF Tc2_Standard.R_TRIG;
	K3:INT;
	K4:INT;
	
	csAxis                 :ARRAY[1..MaxAxes] OF   CS_AxisCtrl;
	fbCy                   :ARRAY[1..MaxCy]    OF   FB_CylinderV2;
    fbRec                 :ARRAY[1..MaxRec]   OF   FB_Rectify;
	fbDustMotor       :ARRAY[1..MaxDust]   OF   CS_DustMoter;


    csCodeTcp:CS_CodeTcp;
    fbCamInTest: MC_CamIn;//主轴与驱动凸轮耦合

//速度模式验证
	MC_ExtSetPointGenDisable: MC_ExtSetPointGenDisable;
	MC_ExtSetPointGenEnable: MC_ExtSetPointGenEnable;
    MC_ExtSetPointGenOut:        Tc2_MC2.ST_McOutputs;
    MC_ExtSetPointGenOut2:        Tc2_MC2.ST_McOutputs;

    tonEStop:                     Tc2_Standard.TON;
   
  fbAnSetp1Moter  : CS_SetpMoter;
  fbCaSetp1Moter:CS_SetpMoter;
 // fbP4CutElectric_CY   :FB_Electric_CY;   电缸


	mc_Home    :MC_Home;

     fbCoeWrite_GlueFeed:       FB_EcCoeSdoWrite;
     	wEncodeHome                    :WORD:=6;
	test:ARRAY[1..10] OF BOOL;
	bAnReady:BOOL;//正极准备好
	bCaReady:BOOL;//负极准备好
	//fbDataXML       : FB_DataXML;
	rt10:Tc2_Standard.R_TRIG;
	testii:INT:=0;
	
	Code_MES				:ARRAY[1..20]OF  R_TRIG;
	fCode_MES				:ARRAY[1..20]OF  F_TRIG;
	tCode_MES				:ARRAY[1..20]OF  TON;
	
//模切直线电机COE寻址修改参数
	FB_EcCoESdoWrite_AnSEPTATCache : ARRAY[1..4] OF FB_EcCoESdoWrite; //正极极片缓存参数修改
	FB_EcCoESdoWrite_AnDriverDDR : ARRAY[1..4] OF FB_EcCoESdoWrite;	  //正极主驱参数修改
	FB_EcCoESdoWrite_CaSEPTATCache : ARRAY[1..4] OF FB_EcCoESdoWrite; //正极极片缓存参数修改
	FB_EcCoESdoWrite_CaDriverDDR : ARRAY[1..4] OF FB_EcCoESdoWrite;	  //正极主驱参数修改
	
	wSaveCoeCode  :DWORD:=16#65766173;    //电机参数保存
	
	SEPTATCache_fSmoothValue   :ARRAY[1..4] OF REAL;    //隔膜缓存写入参数值
	SEPTATCache_bWriteCoeValue  :ARRAY[1..4] OF BOOL;    //隔膜缓存写入执行	
	SEPTATCache_SavePara  :ARRAY[1..4] OF BOOL;   //隔膜缓存参数保存
	
	DriverDDR_fSmoothValue   :ARRAY[1..4] OF REAL;    //主驱写入参数值
	DriverDDR_bWriteCoeValue  :ARRAY[1..4] OF BOOL;    //主驱写入执行	
	DriverDDR_SavePara  :ARRAY[1..4] OF BOOL;   //主驱参数保存
	
	ExcelRate_R	:R_TRIG;	//Mes读取优报表	xfp20240316
	MTDWtStep: UINT;
	rDoorAlm :ARRAY[1..2]OF R_TRIG;
END_VAR

	aAirAlarm_TON(IN:=NOT I205[5],PT:=T#1S,Q=>);											
R_TRIG_Bt[1](CLK:= stSysState.btnStart OR stSysState.hmiStart);//启动上升沿
R_TRIG_Bt[2](CLK:= stSysState.btnStop  OR  stSysState.hmiStop);//停止上升沿
R_TRIG_Bt[4](CLK:=  stSysState.btnAuto OR  stSysState.hmiAuto);//手自动切换上升沿
R_TRIG_Bt[5](CLK:=  NOT stSysState.btnAuto);
R_TRIG_Bt[6](CLK:=stSysState.btnEstop);
R_TRIG_Bt[7](CLK:=stSysState.btnReset OR  stSysState.hmiReset );
R_TRIG_Bt[8](CLK:=  NOT stSysState.hmiAuto);



IF R_TRIG_Bt[4].Q THEN  //自动
	stSysState.FlgAuto:=TRUE;
	stSysState.FlgManua:=FALSE;
END_IF
IF R_TRIG_Bt[5].Q  OR  R_TRIG_Bt[8].Q   THEN  //手动
	stSysState.FlgAuto:=FALSE;
	stSysState.FlgManua:=TRUE;
	stSysState.bwindow:=FALSE;
END_IF
stSysState.bReset:=R_TRIG_Bt[7].Q  OR  bInitReset    ;  //复位

stSysState.bAnccdstate:= NOT AnAlarm.arrFlowAlarm[8] AND NOT AnAlarm.arrFlowAlarm[14] AND  ((NOT ProductPar.iModeEN.bCcdTcpEN AND NOT ProductPar.iModeEN.bSizeCCDEN  AND 
                         NOT  ProductPar.iModeEN.bChamferCCDEN AND NOT  ProductPar.iModeEN.bCuterCCDEN(* AND NOT  ProductPar.iModeEN.bLineScanCCDEN*)) OR  ProductPar.iModeEN.bP2PartEN);
stSysState.bCaccdstate:= NOT CaAlarm.arrFlowAlarm[8] AND NOT CaAlarm.arrFlowAlarm[14] AND  ((NOT ProductPar.iModeEN.bCcdTcpEN AND NOT ProductPar.iModeEN.bSizeCCDEN  AND 
                         NOT  ProductPar.iModeEN.bChamferCCDEN AND NOT  ProductPar.iModeEN.bCuterCCDEN (*AND NOT  ProductPar.iModeEN.bLineScanCCDEN*)) OR  ProductPar.iModeEN.bP2PartEN);

//////////////////////////////////系统流程///////////////////////
CASE iMainSetp OF 
0://   INIT
    Init();
    stSysState.iMode:=0;
 IF  stSysState.bInitDone THEN
     iMainSetp:=88;	
  END_IF
88://切换手动
  IF  stSysState.FlgManua THEN
	  iMainSetp:=300;
  END_IF
   
 (***********************手动*********************************) 
300:
   stSysState.iMode:=3;
   iMainSetp:=350;  
   
350: 
  	IF  R_TRIG_Bt[1].Q  AND stSysState.FlgAuto THEN  //启动按钮  
		IF stSysState.bAutoCondition THEN
		  stSysState.bwindow:=TRUE;	
	      iMainSetp:=90;
	    END_IF
	END_IF 
	
	IF  stSysState.FlgManua AND TON20.Q THEN  //系统清除
	   iMainSetp:=999;
	END_IF

 90:	
  	IF  R_TRIG_Bt[1].Q  AND stSysState.FlgAuto AND NOT stSysState.bwindow  THEN  //启动按钮  
		IF stSysState.bAutoCondition AND (stSysState.bAnccdstate OR ProductPar.iModeEN.iModeRun=1) AND (stSysState.bCaccdstate OR ProductPar.iModeEN.iModeRun=2) THEN
	      iMainSetp:=100;
	    END_IF
		
	ELSIF stSysState.FlgManua OR  stSysState.btnStop  OR  stSysState.hmiStop   OR   stSysState.bErrorStop OR 
          stSysState.btnEstop OR NOT stSysState.bAnccdstate OR NOT stSysState.bCaccdstate  THEN
		  iMainSetp:=300;
	END_IF 	
	
 (************************自动********************************) 
100:
   stSysState.iMode:=1;
   iMainSetp:=150;  
150:  //系统停止中......
    rtStoping(Clk:=stSysState.FlgManua OR  stSysState.btnStop  OR  stSysState.hmiStop   OR   stSysState.bErrorStop OR stSysState.btnEstop);  //自动中触发手动 停止 按钮  stSysRun.bErrorStop 包括正极和负极
    IF stSysState.FlgManua OR  stSysState.btnStop  OR  stSysState.hmiStop   OR   stSysState.bErrorStop OR stSysState.btnEstop THEN //自动触发停止 rtStoping.Q
		stSysState.Stoping:=TRUE;
		iMainSetp:=160; //
	END_IF;
	
160: //判断停止完成
   	IF  stSysState.bStopFinished  THEN
		AnSys.bStopFinished:=FALSE; 
		CaSys.bStopFinished:=FALSE;
       	stSysState.Stoping:=FALSE;
		IF NOT  stSysState.btnEstop THEN
			iMainSetp:=300; 
		ELSE
			stSysState.bInitDone:=FALSE;
			iMainSetp:=400; 	
		END_IF
	END_IF;
	
 (************************急停********************************) 
400://Stoping
   stSysState.iMode:=4;
    EStop();  
   iMainSetp:=450; 
      
450: //急停跳出 
	IF  NOT  stSysState.btnEstop  THEN  
        tonEStop(IN:=FALSE , PT:=T#50MS );
	    iMainSetp:=0;
    ELSE
         tonEStop(IN:=TRUE , PT:=T#50MS );
         IF  tonEStop.Q THEN
              tonEStop(IN:=FALSE , PT:=T#50MS );
              iMainSetp:=400;   
         END_IF
   	 END_IF

END_CASE


IF   stSysState.btnEstop   THEN  //AND  stSysState.iMode=3
	  iMainSetp:=400;
END_IF



(***************程序调用*********************)



AnPart(iMode:=stSysState.iMode);
CaPart(iMode:=stSysState.iMode);
//	XML();
   Condition();
    MotionBasic();
    CyBasic();
    RecBasic();
     Alarm();
     Pusle();
	 MS_Alarm();
	 Motion_coe();
	 MesCollect();
//PoleData.AnBeltData[1].Meney.SizeResults;

ACTION Alarm:

IF NOT ProductPar.iModeEN.bDoorEN THEN
	IF NOT I206[15] THEN
		aAlarm[49]:=TRUE;//模切通道安全门报警
	END_IF
END_IF



IF R_TRIG_Bt[7].Q THEN
	FOR K1:=1 TO MaxAxes DO 
     arrAxisAlarm[K1]:=  FALSE ;
END_FOR
END_IF
(******************气缸报警*******************)
FOR K1:=1 TO MaxCy DO 
     arrCYOnAlarm[K1]:=  arrCyCtrl[K1] .Status.Error1;
     arrCYOFFAlarm[K1]:=  arrCyCtrl[K1] .Status.Error2;
END_FOR
(******************正极气缸报警*******************)
bAnCYHaveAlarm:=FALSE;
FOR K1:=1 TO 20 DO 
      bAnCYHaveAlarm:=(bAnCYHaveAlarm OR arrCYOnAlarm[K1] OR  arrCYOFFAlarm[K1]) ;
END_FOR
FOR K1:=41 TO 60 DO 
      bAnCYHaveAlarm:=(bAnCYHaveAlarm OR arrCYOnAlarm[K1] OR  arrCYOFFAlarm[K1]) ;
END_FOR
(******************负极气缸报警*******************)
bCaCYHaveAlarm:=FALSE;
FOR K1:=21 TO 40 DO 
      bCaCYHaveAlarm:=(bCaCYHaveAlarm OR arrCYOnAlarm[K1] OR  arrCYOFFAlarm[K1]) ;
END_FOR
FOR K1:=61 TO MaxCy DO 
      bCaCYHaveAlarm:=(bCaCYHaveAlarm OR arrCYOnAlarm[K1] OR  arrCYOFFAlarm[K1]) ;
END_FOR

(******************切刀计数报警*************)
IF ProductPar.AnPar.iMouldCount1>= ProductPar.AnPar.iMouldCountAlarm1 THEN   //正极前模具切刀计数报警
	CuterCountAlarm[1]:=TRUE;
	ELSE
	CuterCountAlarm[1]:=FALSE;	
END_IF
(*IF ProductPar.AnPar.iMouldCount2>= ProductPar.AnPar.iMouldCountAlarm2 THEN   //正极后模具切刀计数报警
	CuterCountAlarm[2]:=TRUE;
	ELSE
	CuterCountAlarm[2]:=FALSE;	
END_IF*)
IF ProductPar.AnPar.iCuterCount>= ProductPar.AnPar.iCuterCountAlarm THEN   //正极裁切切刀计数报警
	CuterCountAlarm[3]:=TRUE;
	ELSE
	CuterCountAlarm[3]:=FALSE;	
END_IF
IF ProductPar.CaPar.iMouldCount1>= ProductPar.CaPar.iMouldCountAlarm1 THEN   //负极前模具切刀计数报警
	CuterCountAlarm[4]:=TRUE;
	ELSE
	CuterCountAlarm[4]:=FALSE;	
END_IF
(*IF ProductPar.CaPar.iMouldCount2>= ProductPar.CaPar.iMouldCountAlarm2 THEN   //负极后模具切刀计数报警
	CuterCountAlarm[5]:=TRUE;
	ELSE
	CuterCountAlarm[5]:=FALSE;	
END_IF*)
IF ProductPar.CaPar.iCuterCount>= ProductPar.CaPar.iCuterCountAlarm THEN   //负极裁切切刀计数报警
	CuterCountAlarm[6]:=TRUE;
	ELSE
	CuterCountAlarm[6]:=FALSE;	
END_IF

IF CuterCountAlarm[1] OR CuterCountAlarm[3] OR CuterCountAlarm[4] OR CuterCountAlarm[6] THEN// OR CuterCountAlarm[2] OR CuterCountAlarm[5]
	b_lifetime:=TRUE;
	ELSE
	b_lifetime:=FALSE;	
END_IF

IF ProductPar.AnPar.iCuterCount>= ProductPar.AnPar.iCuterCountWarning THEN    //正极裁切切刀计数预警
	CuterCountAlarm[7]:=TRUE;
	ELSE
	CuterCountAlarm[7]:=FALSE;	
END_IF
IF ProductPar.CaPar.iCuterCount>= ProductPar.CaPar.iCuterCountWarning THEN   //负极裁切切刀计数预警
	CuterCountAlarm[8]:=TRUE;
	ELSE
	CuterCountAlarm[8]:=FALSE;	
END_IF

(****************轴报警**************)
(*
FOR K1:=1 TO MaxAxes DO 
     arrAxisAlarm[K1]:=  arrAxis[K1] .Status.Error AND  arrAxis[K1] .Status.ErrorID<>16#42A0 OR NOT arrAxisCtrl[K1] .Status.Enabled ;
END_FOR
*)
(****************正极轴报警**************)
bAnAxisHaveAlarm:=FALSE;
FOR K1:=1 TO 15 DO 
		IF K1<>3 AND K1<>4 THEN
				arrAxisAlarm[K1]:=  arrAxis[K1] .Status.Error AND  arrAxis[K1] .Status.ErrorID<>16#42A0  ;//OR NOT arrAxisCtrl[K1] .Status.Enabled
				bAnAxisHaveAlarm:=bAnAxisHaveAlarm OR arrAxisAlarm[K1]  ;//OR arrAxisCtrl[K1] .Status.ErrorLimitSwitch
		END_IF
END_FOR

FOR K1:=18 TO 22 DO 
	  arrAxisAlarm[K1]:=  arrAxis[K1] .Status.Error AND  arrAxis[K1] .Status.ErrorID<>16#42A0  ;//OR NOT arrAxisCtrl[K1] .Status.Enabled
      bAnAxisHaveAlarm:=bAnAxisHaveAlarm OR arrAxisAlarm[K1]  ;//OR arrAxisCtrl[K1] .Status.ErrorLimitSwitch
END_FOR

FOR K1:=50 TO 52 DO 
	  arrAxisAlarm[K1]:=  arrAxis[K1] .Status.Error AND  arrAxis[K1] .Status.ErrorID<>16#42A0  ;//OR NOT arrAxisCtrl[K1] .Status.Enabled
      bAnAxisHaveAlarm:=bAnAxisHaveAlarm OR arrAxisAlarm[K1]  ;//OR arrAxisCtrl[K1] .Status.ErrorLimitSwitch
END_FOR

(****************负极轴报警**************)
bCaAxisHaveAlarm:=FALSE;
FOR K1:=25 TO 39 DO 
		IF K1<>27 AND K1<>28 THEN
				arrAxisAlarm[K1]:=  arrAxis[K1] .Status.Error AND  arrAxis[K1] .Status.ErrorID<>16#42A0  ;//OR NOT arrAxisCtrl[K1] .Status.Enabled
				bCaAxisHaveAlarm:=bCaAxisHaveAlarm OR arrAxisAlarm[K1]  ;//OR arrAxisCtrl[K1] .Status.ErrorLimitSwitch
		END_IF
END_FOR

FOR K1:=42 TO 46 DO 
	  arrAxisAlarm[K1]:=  arrAxis[K1] .Status.Error AND  arrAxis[K1] .Status.ErrorID<>16#42A0  ;//OR NOT arrAxisCtrl[K1] .Status.Enabled
      bCaAxisHaveAlarm:=bCaAxisHaveAlarm OR arrAxisAlarm[K1]  ;//OR arrAxisCtrl[K1] .Status.ErrorLimitSwitch
END_FOR

FOR K1:=56 TO 58 DO
	  arrAxisAlarm[K1]:=  arrAxis[K1] .Status.Error AND  arrAxis[K1] .Status.ErrorID<>16#42A0  ; //OR NOT arrAxisCtrl[K1] .Status.Enabled
      bCaAxisHaveAlarm:=bCaAxisHaveAlarm OR arrAxisAlarm[K1]  ;//OR arrAxisCtrl[K1] .Status.ErrorLimitSwitch
END_FOR

(******************张力报警*******************)
bAnTenHaveAlarm :=FALSE;
bCaTenHaveAlarm :=FALSE;
FOR K1:=1 TO 15 DO 
      bAnTenHaveAlarm:=bAnTenHaveAlarm OR AnAlarm.arrTenAlarm[K1];
	  bCaTenHaveAlarm:=bCaTenHaveAlarm OR CaAlarm.arrTenAlarm[K1];
END_FOR

(******************凸轮报警*******************)
bAnCreatTableHaveAlarm :=FALSE;
bCaCreatTableHaveAlarm :=FALSE;
bAnCamHaveAlarm :=FALSE;
bCaCamHaveAlarm :=FALSE;
FOR K1:=1 TO 30 DO 
      bAnCreatTableHaveAlarm:=bAnCreatTableHaveAlarm OR AnAlarm.arrCreatTableAlarm[K1];
	  bCaCreatTableHaveAlarm:=bCaCreatTableHaveAlarm OR CaAlarm.arrCreatTableAlarm[K1];
	  bAnCamHaveAlarm:=bAnCamHaveAlarm OR AnAlarm.arrCamInAlarm[K1];
	  bCaCamHaveAlarm:=bAnCamHaveAlarm OR CaAlarm.arrCamInAlarm[K1];
END_FOR

(******************齿轮报警*******************)
bAnGearHaveAlarm :=FALSE;
bCaGearHaveAlarm :=FALSE;
FOR K1:=1 TO 25 DO 
      bAnGearHaveAlarm:=bAnGearHaveAlarm OR AnAlarm.arrGearAlarm[K1];
	  bCaGearHaveAlarm:=bCaGearHaveAlarm OR CaAlarm.arrGearAlarm[K1];
END_FOR

(******************流程报警*******************)
bAnFlowHaveAlarm :=FALSE;
bCaFlowHaveAlarm :=FALSE;
FOR K1:=1 TO 50 DO 
      bAnFlowHaveAlarm:=bAnFlowHaveAlarm OR AnAlarm.arrFlowAlarm[K1];
	  bCaFlowHaveAlarm:=bCaFlowHaveAlarm OR CaAlarm.arrFlowAlarm[K1];
END_FOR

